# B&R Automation Studio project RobotLineDemo
Automation Studio 6.5.3.11; technology packages: mappMotion 6.9.1, OpcUaCs 6.8.0

## Configuration Config1

CPU 5APC4100.TGL4-000, AutomationRuntime 6.8.1, Build 11.3.0

### Task classes (Cpu.sw)
```
Cyclic#1 (cycle 4000 us, tolerance 0 us):
  MovePrg <- Tasks.MovePrg.prg
Cyclic#2:
  Override <- Tasks.Override.prg
DataObjects: McAcpSys
NcDataObjects: McDriveLog
Binaries: McAcpSim, udbdef, McMechSys, FWRules, McAcpDrv, TCData, Config_19, Config_18, Config_17, Config_16, Config_15, Config_14, arconfig, Config_12, Config_11, Config_10, Config_13, Config_1, ConvAxes, User, Config_4, asfw, iomap, Config_24, Config_23, Config_22, Config_21, UaCsConfig, Config_2, ashwd, Hierarchy, Config_7, ToolGeo, ToolDyn, Config_5, Common, Config, ashwac, sysconf, Config_20, Config_8, ProdLoad1, TrkPaths, Config_9, Config_3, Config_6, BRRole, Config_25
Libraries: MpBase, McBase, MpAxis, McAcpAx, McPathGen, McAxGroup, McAxis, McProgInt, McTrkPath, MpRobotics, ArSvcReg, UaCore, AsIecCon, UaCoal, powerlnk, astime, runtime, fileio, AsIOAcc, SYS_LIB, AsArProf, DataObj, UaCoalPrv, AsIO, brsystem, AsMem, AsIoTrc, AsEPL
```

### Hardware
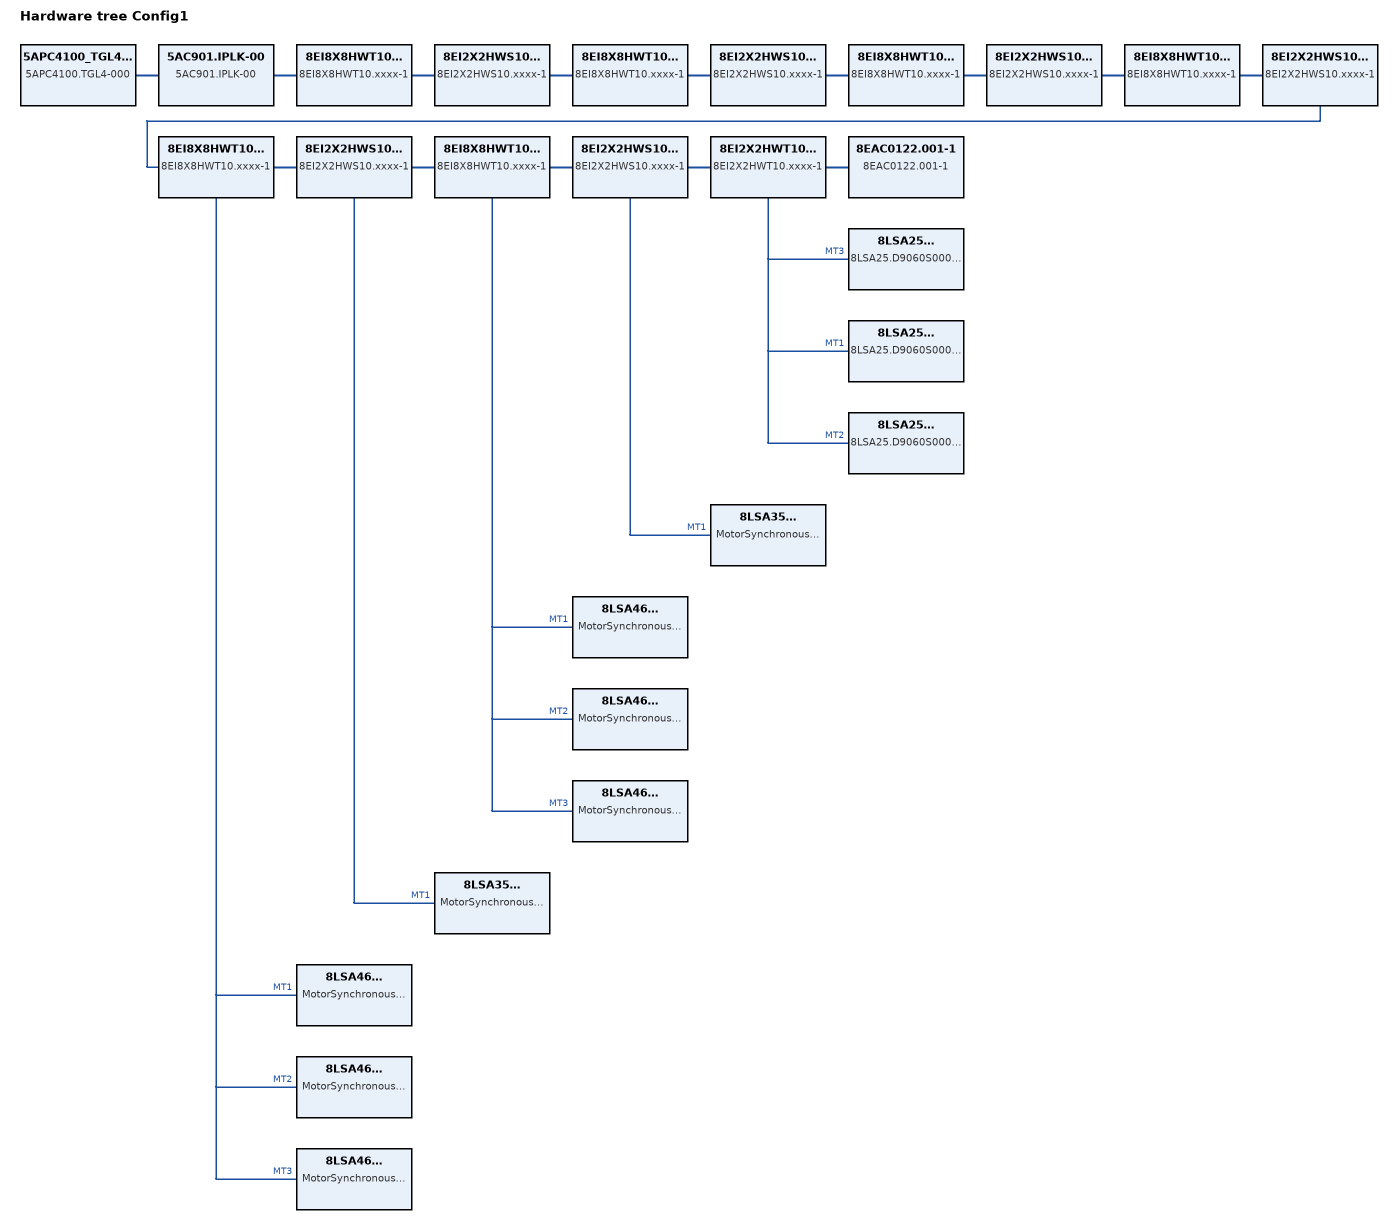
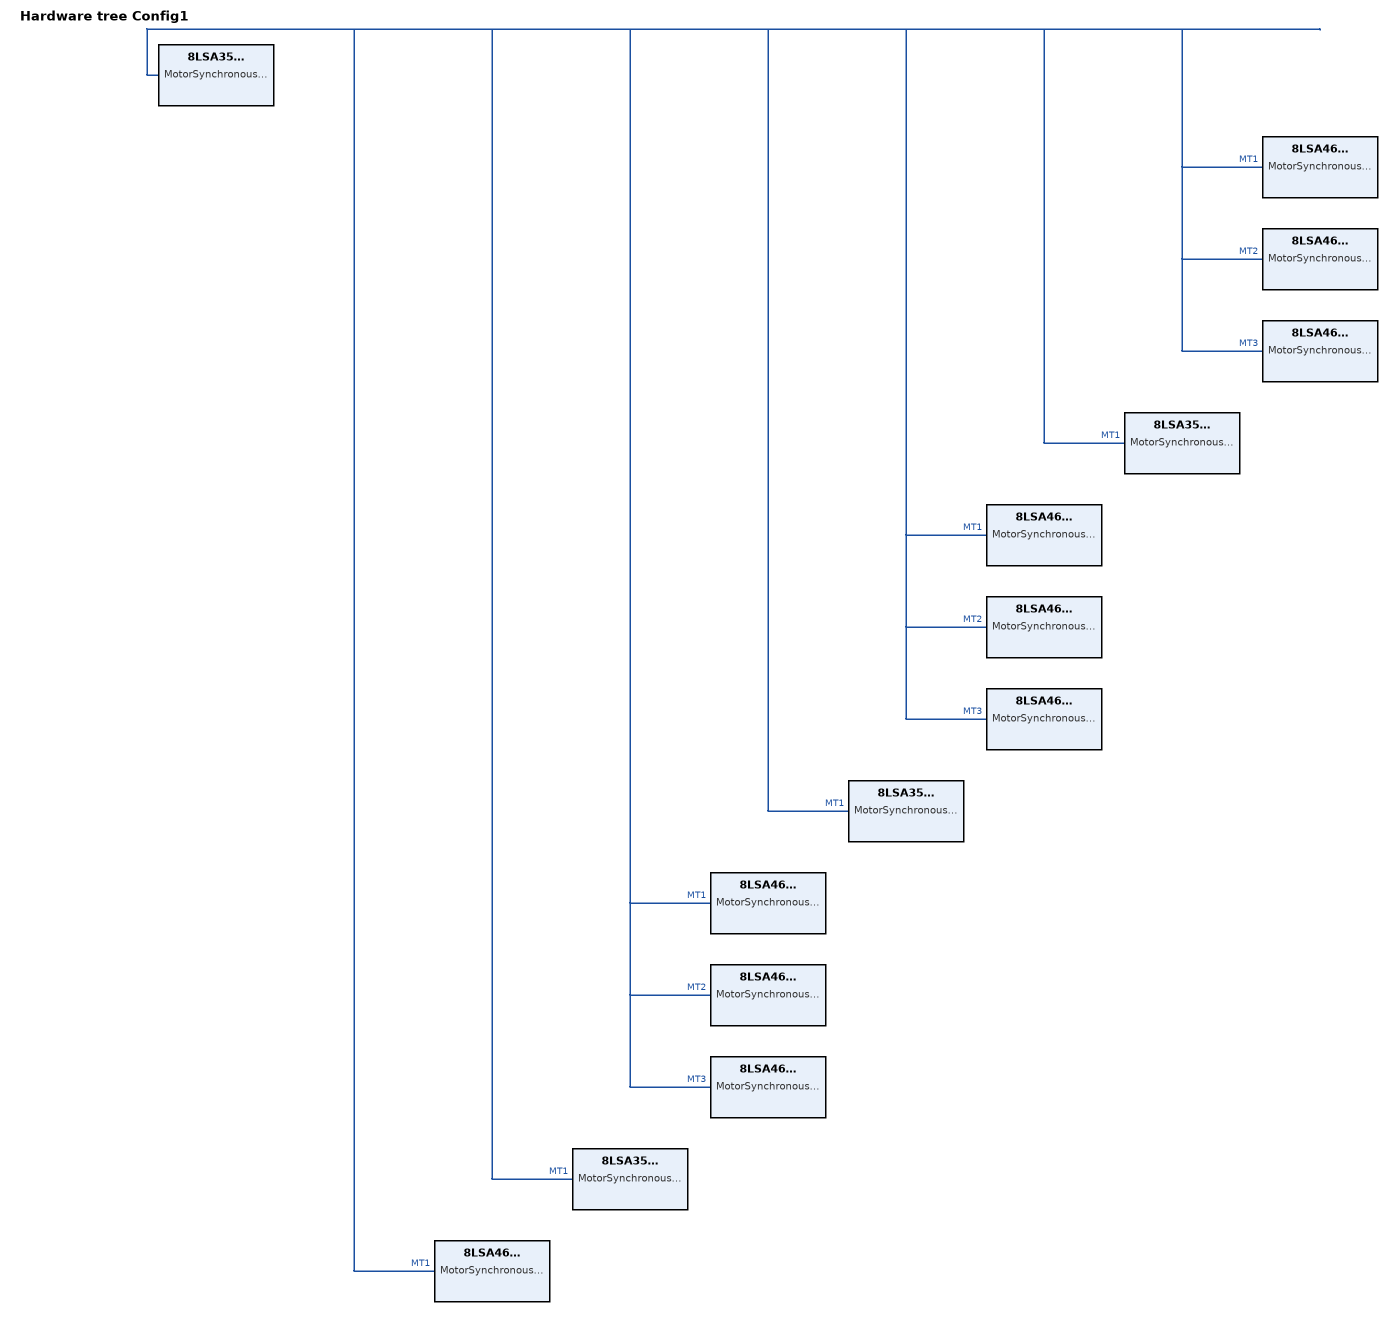
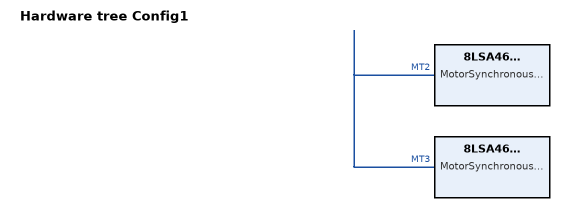
```
5AC901.IPLK-00 : 5AC901.IPLK-00 v2.1.0.0  [SS -> 5APC4100_TGL4_000.SS2]
  Connector IF1:
    EplNatSubnet = 192.168.102.0
5APC4100_TGL4_000 : 5APC4100.TGL4-000 v1.3.1.0
  Connector IF3:
    AssignedOperatingSystem = ARemb
    ActivateDevice = 1
    HostName = laimighoferp-apc4100
    Mode = Manual
    InternetAddress = 172.30.13.10
  Connector IF4:
    AssignedOperatingSystem = ARemb
    ActivateDevice = 1
    HostName = laimighoferp-apc4100
  Connector IF5:
    AssignedOperatingSystem = ARemb
    ActivateDevice = 1
    HostName = laimighoferp-apc4100
  Connector IF6:
    AssignedOperatingSystem = ARemb
    ActivateDevice = 1
    HostName = laimighoferp-apc4100
  Connector IF7:
    AssignedOperatingSystem = ARemb
  Connector IF8:
    AssignedOperatingSystem = ARemb
  Connector IF9:
    AssignedOperatingSystem = ARemb
  Connector IF10:
    AssignedOperatingSystem = ARemb
  Connector IF11:
    AssignedOperatingSystem = ARemb
  Connector IF12:
    AssignedOperatingSystem = ARemb
  ConfigurationID = RobotLineDemoInterpack_Config1
  Simulation = 1
  SimulationIPAddress = 127.0.0.3
  Cyclic1Duration = 4000
  Cyclic1Tolerance = 0
  FileDevice1
  FileDeviceName1 = USER
  FileDevicePath1 = USER_PATH
  FileDevice2
  FileDeviceName2 = CNC_PrgDir
  FileDevicePath2 = USER_PATH/MotionPrg
  FileDevice3
  FileDeviceName3 = Scene
  FileDevicePath3 = USER_PATH/Scenes  // ../../../../../../Logical/Scene/Scenes
  TimeZone = 140
  EthernetHostName = laimighoferp-apc4100
  EthernetDefaultGateway = 172.30.13.1
  ActivateWebServer = 1
  WebServerProtocol = 1
  ActivateSdm = 1
8EAC0122.001-1 : 8EAC0122.001-1 v3.0.0.0  [SS -> 8EI2X2HWT10.xxxx-1.SS1]
8EI2X2HWS10.xxxx-1-QC_D4r1100R_1 : 8EI2X2HWS10.xxxx-1 v2.4.0.0 (NodeNumber=2)  [PLK1 -> 8EI8X8HWT10.xxxx-1-Q1-Q2-Q3_D4r1100R_1.PLK2 [Cable Type=PowerlinkCable, Length=10, Version=1.0.0.3]; PLK2 -> 8EI8X8HWT10.xxxx-1-Q1-Q2-Q3_D4r1100R_2.PLK1 [Cable Type=PowerlinkCable, Length=10, Version=1.0.0.3]]
  DriveConfiguration/Module:
    ActivateACOPOSSimulationOnPLC = 1
  DriveConfiguration/Encoder/EncoderX41:
    InterfaceType = EnDat
  DriveConfiguration/Channel[1]/RealAxis:
    AxisReference = gAxisQC_D4r1100R_1
  DriveConfiguration/Channel[1]/RealAxis/MechanicalElements/Gearbox:
    InputIsReadOnly = 1
    Input = 10
    OutputIsReadOnly = 1
  DriveConfiguration/Channel[1]/RealAxis/MechanicalElements/RotaryToLinearTransformation:
    ReferenceDistanceIsReadOnly = 1
    ReferenceDistance = 360
  DriveConfiguration/Channel[1]/RealAxis/Controller:
    ModeIsReadOnly = 1
    Mode = PositionControllerWithTorqueFeedForward
  DriveConfiguration/Channel[1]/RealAxis/Controller/Mode/Position:
    ProportionalGainIsReadOnly = 1
    ProportionalGain = 25.0
    IntegrationTimeIsReadOnly = 1
  DriveConfiguration/Channel[1]/RealAxis/Controller/Mode/Speed:
    ProportionalGainIsReadOnly = 1
    ProportionalGain = 1.3
    IntegrationTimeIsReadOnly = 1
    FilterTimeIsReadOnly = 1
  DriveConfiguration/Channel[1]/RealAxis/Controller/Mode:
    FeedForwardIsReadOnly = 1
    FeedForward = CyclicValueFromAxesGroup
  DriveConfiguration/Channel[1]/RealAxis/Controller/Mode/LoopFilters:
    LoopFilterXIsReadOnly = 1
  DriveConfiguration/Channel[1]/RealAxis/Homing:
    Mode = Absolute
    RestorePositionVariable = 
  DriveConfiguration/Channel[1]/RealAxis/StopReaction:
    DriveError = CyclicDecelerationFromAxesGroup
  DriveConfiguration/Channel[1]/RealAxis/MovementErrorLimits:
    PositionError = 1.0
  DriveConfiguration/Channel[1]/RealAxis:
    JerkFilterIsReadOnly = 1
    JerkFilter = Used
  DriveConfiguration/Channel[1]/RealAxis/JerkFilter:
    JerkTimeMin = 0.07
    JerkTime = 0.07
8EI2X2HWS10.xxxx-1-QC_D4r1100R_2 : 8EI2X2HWS10.xxxx-1 v2.4.0.0 (NodeNumber=4)  [PLK1 -> 8EI8X8HWT10.xxxx-1-Q1-Q2-Q3_D4r1100R_2.PLK2 [Cable Type=PowerlinkCable, Length=10, Version=1.0.0.3]; PLK2 -> 8EI8X8HWT10.xxxx-1-Q1-Q2-Q3_D4r1100R_3.PLK1 [Cable Type=PowerlinkCable, Length=10, Version=1.0.0.3]]
  DriveConfiguration/Module:
    ActivateACOPOSSimulationOnPLC = 1
  DriveConfiguration/Encoder/EncoderX41:
    InterfaceType = EnDat
  DriveConfiguration/Channel[1]/RealAxis:
    AxisReference = gAxisQC_D4r1100R_2
  DriveConfiguration/Channel[1]/RealAxis/MechanicalElements/Gearbox:
    InputIsReadOnly = 1
    Input = 10
    OutputIsReadOnly = 1
  DriveConfiguration/Channel[1]/RealAxis/MechanicalElements/RotaryToLinearTransformation:
    ReferenceDistanceIsReadOnly = 1
    ReferenceDistance = 360
  DriveConfiguration/Channel[1]/RealAxis/Controller:
    ModeIsReadOnly = 1
    Mode = PositionControllerWithTorqueFeedForward
  DriveConfiguration/Channel[1]/RealAxis/Controller/Mode/Position:
    ProportionalGainIsReadOnly = 1
    ProportionalGain = 25.0
    IntegrationTimeIsReadOnly = 1
  DriveConfiguration/Channel[1]/RealAxis/Controller/Mode/Speed:
    ProportionalGainIsReadOnly = 1
    ProportionalGain = 1.3
    IntegrationTimeIsReadOnly = 1
    FilterTimeIsReadOnly = 1
  DriveConfiguration/Channel[1]/RealAxis/Controller/Mode:
    FeedForwardIsReadOnly = 1
    FeedForward = CyclicValueFromAxesGroup
  DriveConfiguration/Channel[1]/RealAxis/Controller/Mode/LoopFilters:
    LoopFilterXIsReadOnly = 1
  DriveConfiguration/Channel[1]/RealAxis/Homing:
    Mode = Absolute
    RestorePositionVariable = 
  DriveConfiguration/Channel[1]/RealAxis/StopReaction:
    DriveError = CyclicDecelerationFromAxesGroup
  DriveConfiguration/Channel[1]/RealAxis/MovementErrorLimits:
    PositionError = 1.0
  DriveConfiguration/Channel[1]/RealAxis:
    JerkFilterIsReadOnly = 1
    JerkFilter = Used
  DriveConfiguration/Channel[1]/RealAxis/JerkFilter:
    JerkTimeMin = 0.07
    JerkTime = 0.07
8EI2X2HWS10.xxxx-1-QC_D4r1100R_3 : 8EI2X2HWS10.xxxx-1 v2.4.0.0 (NodeNumber=6)  [PLK1 -> 8EI8X8HWT10.xxxx-1-Q1-Q2-Q3_D4r1100R_3.PLK2 [Cable Type=PowerlinkCable, Length=10, Version=1.0.0.3]; PLK2 -> 8EI8X8HWT10.xxxx-1-Q1-Q2-Q3_D4r1100R_4.PLK1 [Cable Type=PowerlinkCable, Length=10, Version=1.0.0.3]]
  DriveConfiguration/Module:
    ActivateACOPOSSimulationOnPLC = 1
  DriveConfiguration/Encoder/EncoderX41:
    InterfaceType = EnDat
  DriveConfiguration/Channel[1]/RealAxis:
    AxisReference = gAxisQC_D4r1100R_3
  DriveConfiguration/Channel[1]/RealAxis/MechanicalElements/Gearbox:
    InputIsReadOnly = 1
    Input = 10
    OutputIsReadOnly = 1
  DriveConfiguration/Channel[1]/RealAxis/MechanicalElements/RotaryToLinearTransformation:
    ReferenceDistanceIsReadOnly = 1
    ReferenceDistance = 360
  DriveConfiguration/Channel[1]/RealAxis/Controller:
    ModeIsReadOnly = 1
    Mode = PositionControllerWithTorqueFeedForward
  DriveConfiguration/Channel[1]/RealAxis/Controller/Mode/Position:
    ProportionalGainIsReadOnly = 1
    ProportionalGain = 25.0
    IntegrationTimeIsReadOnly = 1
  DriveConfiguration/Channel[1]/RealAxis/Controller/Mode/Speed:
    ProportionalGainIsReadOnly = 1
    ProportionalGain = 1.3
    IntegrationTimeIsReadOnly = 1
    FilterTimeIsReadOnly = 1
  DriveConfiguration/Channel[1]/RealAxis/Controller/Mode:
    FeedForwardIsReadOnly = 1
    FeedForward = CyclicValueFromAxesGroup
  DriveConfiguration/Channel[1]/RealAxis/Controller/Mode/LoopFilters:
    LoopFilterXIsReadOnly = 1
  DriveConfiguration/Channel[1]/RealAxis/Homing:
    Mode = Absolute
    RestorePositionVariable = 
  DriveConfiguration/Channel[1]/RealAxis/StopReaction:
    DriveError = CyclicDecelerationFromAxesGroup
  DriveConfiguration/Channel[1]/RealAxis/MovementErrorLimits:
    PositionError = 1.0
  DriveConfiguration/Channel[1]/RealAxis:
    JerkFilterIsReadOnly = 1
    JerkFilter = Used
  DriveConfiguration/Channel[1]/RealAxis/JerkFilter:
    JerkTimeMin = 0.07
    JerkTime = 0.07
8EI2X2HWS10.xxxx-1-QC_D4r1100R_4 : 8EI2X2HWS10.xxxx-1 v2.4.0.0 (NodeNumber=8)  [PLK1 -> 8EI8X8HWT10.xxxx-1-Q1-Q2-Q3_D4r1100R_4.PLK2 [Cable Type=PowerlinkCable, Length=10, Version=1.0.0.3]; PLK2 -> 8EI8X8HWT10.xxxx-1-Q1-Q2-Q3_D4r1100R_5.PLK1 [Cable Type=PowerlinkCable, Length=10, Version=1.0.0.3]]
  DriveConfiguration/Module:
    ActivateACOPOSSimulationOnPLC = 1
  DriveConfiguration/Encoder/EncoderX41:
    InterfaceType = EnDat
  DriveConfiguration/Channel[1]/RealAxis:
    AxisReference = gAxisQC_D4r1100R_4
  DriveConfiguration/Channel[1]/RealAxis/MechanicalElements/Gearbox:
    InputIsReadOnly = 1
    Input = 10
    OutputIsReadOnly = 1
  DriveConfiguration/Channel[1]/RealAxis/MechanicalElements/RotaryToLinearTransformation:
    ReferenceDistanceIsReadOnly = 1
    ReferenceDistance = 360
  DriveConfiguration/Channel[1]/RealAxis/Controller:
    ModeIsReadOnly = 1
    Mode = PositionControllerWithTorqueFeedForward
  DriveConfiguration/Channel[1]/RealAxis/Controller/Mode/Position:
    ProportionalGainIsReadOnly = 1
    ProportionalGain = 25.0
    IntegrationTimeIsReadOnly = 1
  DriveConfiguration/Channel[1]/RealAxis/Controller/Mode/Speed:
    ProportionalGainIsReadOnly = 1
    ProportionalGain = 1.3
    IntegrationTimeIsReadOnly = 1
    FilterTimeIsReadOnly = 1
  DriveConfiguration/Channel[1]/RealAxis/Controller/Mode:
    FeedForwardIsReadOnly = 1
    FeedForward = CyclicValueFromAxesGroup
  DriveConfiguration/Channel[1]/RealAxis/Controller/Mode/LoopFilters:
    LoopFilterXIsReadOnly = 1
  DriveConfiguration/Channel[1]/RealAxis/Homing:
    Mode = Absolute
    RestorePositionVariable = 
  DriveConfiguration/Channel[1]/RealAxis/StopReaction:
    DriveError = CyclicDecelerationFromAxesGroup
  DriveConfiguration/Channel[1]/RealAxis/MovementErrorLimits:
    PositionError = 1.0
  DriveConfiguration/Channel[1]/RealAxis:
    JerkFilterIsReadOnly = 1
    JerkFilter = Used
  DriveConfiguration/Channel[1]/RealAxis/JerkFilter:
    JerkTimeMin = 0.07
    JerkTime = 0.07
8EI2X2HWS10.xxxx-1-QC_D4r1100R_5 : 8EI2X2HWS10.xxxx-1 v2.4.0.0 (NodeNumber=10)  [PLK1 -> 8EI8X8HWT10.xxxx-1-Q1-Q2-Q3_D4r1100R_5.PLK2 [Cable Type=PowerlinkCable, Length=10, Version=1.0.0.3]; PLK2 -> 8EI8X8HWT10.xxxx-1-Q1-Q2-Q3_D4r1100R_6.PLK1 [Cable Type=PowerlinkCable, Length=10, Version=1.0.0.3]]
  DriveConfiguration/Module:
    ActivateACOPOSSimulationOnPLC = 1
  DriveConfiguration/Encoder/EncoderX41:
    InterfaceType = EnDat
  DriveConfiguration/Channel[1]/RealAxis:
    AxisReference = gAxisQC_D4r1100R_5
  DriveConfiguration/Channel[1]/RealAxis/MechanicalElements/Gearbox:
    InputIsReadOnly = 1
    Input = 10
    OutputIsReadOnly = 1
  DriveConfiguration/Channel[1]/RealAxis/MechanicalElements/RotaryToLinearTransformation:
    ReferenceDistanceIsReadOnly = 1
    ReferenceDistance = 360
  DriveConfiguration/Channel[1]/RealAxis/Controller:
    ModeIsReadOnly = 1
    Mode = PositionControllerWithTorqueFeedForward
  DriveConfiguration/Channel[1]/RealAxis/Controller/Mode/Position:
    ProportionalGainIsReadOnly = 1
    ProportionalGain = 25.0
    IntegrationTimeIsReadOnly = 1
  DriveConfiguration/Channel[1]/RealAxis/Controller/Mode/Speed:
    ProportionalGainIsReadOnly = 1
    ProportionalGain = 1.3
    IntegrationTimeIsReadOnly = 1
    FilterTimeIsReadOnly = 1
  DriveConfiguration/Channel[1]/RealAxis/Controller/Mode:
    FeedForwardIsReadOnly = 1
    FeedForward = CyclicValueFromAxesGroup
  DriveConfiguration/Channel[1]/RealAxis/Controller/Mode/LoopFilters:
    LoopFilterXIsReadOnly = 1
  DriveConfiguration/Channel[1]/RealAxis/Homing:
    Mode = Absolute
    RestorePositionVariable = 
  DriveConfiguration/Channel[1]/RealAxis/StopReaction:
    DriveError = CyclicDecelerationFromAxesGroup
  DriveConfiguration/Channel[1]/RealAxis/MovementErrorLimits:
    PositionError = 1.0
  DriveConfiguration/Channel[1]/RealAxis:
    JerkFilterIsReadOnly = 1
    JerkFilter = Used
  DriveConfiguration/Channel[1]/RealAxis/JerkFilter:
    JerkTimeMin = 0.07
    JerkTime = 0.07
8EI2X2HWS10.xxxx-1-QC_D4r1100R_6 : 8EI2X2HWS10.xxxx-1 v2.4.0.0 (NodeNumber=12)  [PLK1 -> 8EI8X8HWT10.xxxx-1-Q1-Q2-Q3_D4r1100R_6.PLK2 [Cable Type=PowerlinkCable, Length=10, Version=1.0.0.3]; PLK2 -> 8EI2X2HWT10.xxxx-1.PLK1 [Cable Type=PowerlinkCable, Length=10, Version=1.0.0.3]]
  DriveConfiguration/Module:
    ActivateACOPOSSimulationOnPLC = 1
  DriveConfiguration/Encoder/EncoderX41:
    InterfaceType = EnDat
  DriveConfiguration/Channel[1]/RealAxis:
    AxisReference = gAxisQC_D4r1100R_6
  DriveConfiguration/Channel[1]/RealAxis/MechanicalElements/Gearbox:
    InputIsReadOnly = 1
    Input = 10
    OutputIsReadOnly = 1
  DriveConfiguration/Channel[1]/RealAxis/MechanicalElements/RotaryToLinearTransformation:
    ReferenceDistanceIsReadOnly = 1
    ReferenceDistance = 360
  DriveConfiguration/Channel[1]/RealAxis/Controller:
    ModeIsReadOnly = 1
    Mode = PositionControllerWithTorqueFeedForward
  DriveConfiguration/Channel[1]/RealAxis/Controller/Mode/Position:
    ProportionalGainIsReadOnly = 1
    ProportionalGain = 25.0
    IntegrationTimeIsReadOnly = 1
  DriveConfiguration/Channel[1]/RealAxis/Controller/Mode/Speed:
    ProportionalGainIsReadOnly = 1
    ProportionalGain = 1.3
    IntegrationTimeIsReadOnly = 1
    FilterTimeIsReadOnly = 1
  DriveConfiguration/Channel[1]/RealAxis/Controller/Mode:
    FeedForwardIsReadOnly = 1
    FeedForward = CyclicValueFromAxesGroup
  DriveConfiguration/Channel[1]/RealAxis/Controller/Mode/LoopFilters:
    LoopFilterXIsReadOnly = 1
  DriveConfiguration/Channel[1]/RealAxis/Homing:
    Mode = Absolute
    RestorePositionVariable = 
  DriveConfiguration/Channel[1]/RealAxis/StopReaction:
    DriveError = CyclicDecelerationFromAxesGroup
  DriveConfiguration/Channel[1]/RealAxis/MovementErrorLimits:
    PositionError = 1.0
  DriveConfiguration/Channel[1]/RealAxis:
    JerkFilterIsReadOnly = 1
    JerkFilter = Used
  DriveConfiguration/Channel[1]/RealAxis/JerkFilter:
    JerkTimeMin = 0.07
    JerkTime = 0.07
8EI2X2HWT10.xxxx-1 : 8EI2X2HWT10.xxxx-1 v2.4.0.0 (NodeNumber=13)  [PLK1 -> 8EI2X2HWS10.xxxx-1-QC_D4r1100R_6.PLK2 [Cable Type=PowerlinkCable, Length=10, Version=1.0.0.3]; MT2 -> 8LSA25.D9060S000-3_b.MT; MT3 -> 8LSA25.D9060S000-3.MT]
  DriveConfiguration/Module:
    ActivateACOPOSSimulationOnPLC = 1
  DriveConfiguration/Channel[1]/RealAxis:
    AxisReference = gAxis_Conveyor_1
  DriveConfiguration/Channel[2]/RealAxis:
    AxisReference = gAxis_Conveyor_2
8EI8X8HWT10.xxxx-1-Q1-Q2-Q3_D4r1100R_1 : 8EI8X8HWT10.xxxx-1 v2.4.0.0 (NodeNumber=1)  [PLK1 -> 5AC901.IPLK-00.IF1 [Cable Type=PowerlinkCable, Length=10, Version=1.0.0.3]; PLK2 -> 8EI2X2HWS10.xxxx-1-QC_D4r1100R_1.PLK1 [Cable Type=PowerlinkCable, Length=10, Version=1.0.0.3]; MT2 -> 8LSA46.DB060S200-3-Q2_D4r1100R_1.MT; MT3 -> 8LSA46.DB060S200-3-Q3_D4r1100R_1.MT]
  DriveConfiguration/Module:
    ActivateACOPOSSimulationOnPLC = 1
  DriveConfiguration/Encoder/EncoderX41:
    InterfaceType = EnDat
  DriveConfiguration/Encoder/EncoderX42:
    InterfaceType = EnDat
  DriveConfiguration/Encoder/EncoderX43:
    InterfaceType = EnDat
  DriveConfiguration/Channel[1]/RealAxis:
    AxisReference = gAxisQ1_D4r1100R_1
  DriveConfiguration/Channel[1]/RealAxis/MechanicalElements/Gearbox:
    InputIsReadOnly = 1
    Input = 77
    OutputIsReadOnly = 1
    Output = 2
  DriveConfiguration/Channel[1]/RealAxis/MechanicalElements/RotaryToLinearTransformation:
    ReferenceDistanceIsReadOnly = 1
    ReferenceDistance = 360
  DriveConfiguration/Channel[1]/RealAxis/Controller:
    ModeIsReadOnly = 1
    Mode = PositionControllerWithTorqueFeedForward
  DriveConfiguration/Channel[1]/RealAxis/Controller/Mode/Position:
    ProportionalGainIsReadOnly = 1
    ProportionalGain = 15.0
    IntegrationTimeIsReadOnly = 1
  DriveConfiguration/Channel[1]/RealAxis/Controller/Mode/Speed:
    ProportionalGainIsReadOnly = 1
    ProportionalGain = 8.0
    IntegrationTimeIsReadOnly = 1
    FilterTimeIsReadOnly = 1
  DriveConfiguration/Channel[1]/RealAxis/Controller/Mode:
    FeedForwardIsReadOnly = 1
    FeedForward = CyclicValueFromAxesGroup
  DriveConfiguration/Channel[1]/RealAxis/Controller/Mode/LoopFilters:
    LoopFilterXIsReadOnly = 1
  DriveConfiguration/Channel[1]/RealAxis/Homing:
    Mode = AbsoluteCorrection
    RestorePositionVariable = 
  DriveConfiguration/Channel[1]/RealAxis/StopReaction:
    DriveError = CyclicDecelerationFromAxesGroup
  DriveConfiguration/Channel[1]/RealAxis/MovementErrorLimits:
    PositionError = 0.5
  DriveConfiguration/Channel[1]/RealAxis:
    JerkFilterIsReadOnly = 1
    JerkFilter = Used
  DriveConfiguration/Channel[1]/RealAxis/JerkFilter:
    JerkTimeMin = 0.07
    JerkTime = 0.07
  DriveConfiguration/Channel[2]/RealAxis:
    AxisReference = gAxisQ2_D4r1100R_1
  DriveConfiguration/Channel[2]/RealAxis/MechanicalElements/Gearbox:
    InputIsReadOnly = 1
    Input = 77
    OutputIsReadOnly = 1
    Output = 2
  DriveConfiguration/Channel[2]/RealAxis/MechanicalElements/RotaryToLinearTransformation:
    ReferenceDistanceIsReadOnly = 1
    ReferenceDistance = 360
  DriveConfiguration/Channel[2]/RealAxis/Controller:
    ModeIsReadOnly = 1
    Mode = PositionControllerWithTorqueFeedForward
  DriveConfiguration/Channel[2]/RealAxis/Controller/Mode/Position:
    ProportionalGainIsReadOnly = 1
    ProportionalGain = 15.0
    IntegrationTimeIsReadOnly = 1
  DriveConfiguration/Channel[2]/RealAxis/Controller/Mode/Speed:
    ProportionalGainIsReadOnly = 1
    ProportionalGain = 8.0
    IntegrationTimeIsReadOnly = 1
    FilterTimeIsReadOnly = 1
  DriveConfiguration/Channel[2]/RealAxis/Controller/Mode:
    FeedForwardIsReadOnly = 1
    FeedForward = CyclicValueFromAxesGroup
  DriveConfiguration/Channel[2]/RealAxis/Controller/Mode/LoopFilters:
    LoopFilterXIsReadOnly = 1
  DriveConfiguration/Channel[2]/RealAxis/Homing:
    Mode = AbsoluteCorrection
    RestorePositionVariable = 
  DriveConfiguration/Channel[2]/RealAxis/StopReaction:
    DriveError = CyclicDecelerationFromAxesGroup
  DriveConfiguration/Channel[2]/RealAxis/MovementErrorLimits:
    PositionError = 0.5
  DriveConfiguration/Channel[2]/RealAxis:
    JerkFilterIsReadOnly = 1
    JerkFilter = Used
  DriveConfiguration/Channel[2]/RealAxis/JerkFilter:
    JerkTimeMin = 0.07
    JerkTime = 0.07
  DriveConfiguration/Channel[3]/RealAxis:
    AxisReference = gAxisQ3_D4r1100R_1
  DriveConfiguration/Channel[3]/RealAxis/MechanicalElements/Gearbox:
    InputIsReadOnly = 1
    Input = 77
    OutputIsReadOnly = 1
    Output = 2
  DriveConfiguration/Channel[3]/RealAxis/MechanicalElements/RotaryToLinearTransformation:
    ReferenceDistanceIsReadOnly = 1
    ReferenceDistance = 360
  DriveConfiguration/Channel[3]/RealAxis/Controller:
    ModeIsReadOnly = 1
    Mode = PositionControllerWithTorqueFeedForward
  DriveConfiguration/Channel[3]/RealAxis/Controller/Mode/Position:
    ProportionalGainIsReadOnly = 1
    ProportionalGain = 15.0
    IntegrationTimeIsReadOnly = 1
  DriveConfiguration/Channel[3]/RealAxis/Controller/Mode/Speed:
    ProportionalGainIsReadOnly = 1
    ProportionalGain = 8.0
    IntegrationTimeIsReadOnly = 1
    FilterTimeIsReadOnly = 1
  DriveConfiguration/Channel[3]/RealAxis/Controller/Mode:
    FeedForwardIsReadOnly = 1
    FeedForward = CyclicValueFromAxesGroup
  DriveConfiguration/Channel[3]/RealAxis/Controller/Mode/LoopFilters:
    LoopFilterXIsReadOnly = 1
  DriveConfiguration/Channel[3]/RealAxis/Homing:
    Mode = AbsoluteCorrection
    RestorePositionVariable = 
  DriveConfiguration/Channel[3]/RealAxis/StopReaction:
    DriveError = CyclicDecelerationFromAxesGroup
  DriveConfiguration/Channel[3]/RealAxis/MovementErrorLimits:
    PositionError = 0.5
  DriveConfiguration/Channel[3]/RealAxis:
    JerkFilterIsReadOnly = 1
    JerkFilter = Used
  DriveConfiguration/Channel[3]/RealAxis/JerkFilter:
    JerkTimeMin = 0.07
    JerkTime = 0.07
8EI8X8HWT10.xxxx-1-Q1-Q2-Q3_D4r1100R_2 : 8EI8X8HWT10.xxxx-1 v2.4.0.0 (NodeNumber=3)  [PLK1 -> 8EI2X2HWS10.xxxx-1-QC_D4r1100R_1.PLK2 [Cable Type=PowerlinkCable, Length=10, Version=1.0.0.3]; PLK2 -> 8EI2X2HWS10.xxxx-1-QC_D4r1100R_2.PLK1 [Cable Type=PowerlinkCable, Length=10, Version=1.0.0.3]; MT2 -> 8LSA46.DB060S200-3-Q2_D4r1100R_2.MT; MT3 -> 8LSA46.DB060S200-3-Q3_D4r1100R_2.MT]
  DriveConfiguration/Module:
    ActivateACOPOSSimulationOnPLC = 1
  DriveConfiguration/Encoder/EncoderX41:
    InterfaceType = EnDat
  DriveConfiguration/Encoder/EncoderX42:
    InterfaceType = EnDat
  DriveConfiguration/Encoder/EncoderX43:
    InterfaceType = EnDat
  DriveConfiguration/Channel[1]/RealAxis:
    AxisReference = gAxisQ1_D4r1100R_2
  DriveConfiguration/Channel[1]/RealAxis/MechanicalElements/Gearbox:
    InputIsReadOnly = 1
    Input = 77
    OutputIsReadOnly = 1
    Output = 2
  DriveConfiguration/Channel[1]/RealAxis/MechanicalElements/RotaryToLinearTransformation:
    ReferenceDistanceIsReadOnly = 1
    ReferenceDistance = 360
  DriveConfiguration/Channel[1]/RealAxis/Controller:
    ModeIsReadOnly = 1
    Mode = PositionControllerWithTorqueFeedForward
  DriveConfiguration/Channel[1]/RealAxis/Controller/Mode/Position:
    ProportionalGainIsReadOnly = 1
    ProportionalGain = 15.0
    IntegrationTimeIsReadOnly = 1
  DriveConfiguration/Channel[1]/RealAxis/Controller/Mode/Speed:
    ProportionalGainIsReadOnly = 1
    ProportionalGain = 8.0
    IntegrationTimeIsReadOnly = 1
    FilterTimeIsReadOnly = 1
  DriveConfiguration/Channel[1]/RealAxis/Controller/Mode:
    FeedForwardIsReadOnly = 1
    FeedForward = CyclicValueFromAxesGroup
  DriveConfiguration/Channel[1]/RealAxis/Controller/Mode/LoopFilters:
    LoopFilterXIsReadOnly = 1
  DriveConfiguration/Channel[1]/RealAxis/Homing:
    Mode = AbsoluteCorrection
    RestorePositionVariable = 
  DriveConfiguration/Channel[1]/RealAxis/StopReaction:
    DriveError = CyclicDecelerationFromAxesGroup
  DriveConfiguration/Channel[1]/RealAxis/MovementErrorLimits:
    PositionError = 0.5
  DriveConfiguration/Channel[1]/RealAxis:
    JerkFilterIsReadOnly = 1
    JerkFilter = Used
  DriveConfiguration/Channel[1]/RealAxis/JerkFilter:
    JerkTimeMin = 0.07
    JerkTime = 0.07
  DriveConfiguration/Channel[2]/RealAxis:
    AxisReference = gAxisQ2_D4r1100R_2
  DriveConfiguration/Channel[2]/RealAxis/MechanicalElements/Gearbox:
    InputIsReadOnly = 1
    Input = 77
    OutputIsReadOnly = 1
    Output = 2
  DriveConfiguration/Channel[2]/RealAxis/MechanicalElements/RotaryToLinearTransformation:
    ReferenceDistanceIsReadOnly = 1
    ReferenceDistance = 360
  DriveConfiguration/Channel[2]/RealAxis/Controller:
    ModeIsReadOnly = 1
    Mode = PositionControllerWithTorqueFeedForward
  DriveConfiguration/Channel[2]/RealAxis/Controller/Mode/Position:
    ProportionalGainIsReadOnly = 1
    ProportionalGain = 15.0
    IntegrationTimeIsReadOnly = 1
  DriveConfiguration/Channel[2]/RealAxis/Controller/Mode/Speed:
    ProportionalGainIsReadOnly = 1
    ProportionalGain = 8.0
    IntegrationTimeIsReadOnly = 1
    FilterTimeIsReadOnly = 1
  DriveConfiguration/Channel[2]/RealAxis/Controller/Mode:
    FeedForwardIsReadOnly = 1
    FeedForward = CyclicValueFromAxesGroup
  DriveConfiguration/Channel[2]/RealAxis/Controller/Mode/LoopFilters:
    LoopFilterXIsReadOnly = 1
  DriveConfiguration/Channel[2]/RealAxis/Homing:
    Mode = AbsoluteCorrection
    RestorePositionVariable = 
  DriveConfiguration/Channel[2]/RealAxis/StopReaction:
    DriveError = CyclicDecelerationFromAxesGroup
  DriveConfiguration/Channel[2]/RealAxis/MovementErrorLimits:
    PositionError = 0.5
  DriveConfiguration/Channel[2]/RealAxis:
    JerkFilterIsReadOnly = 1
    JerkFilter = Used
  DriveConfiguration/Channel[2]/RealAxis/JerkFilter:
    JerkTimeMin = 0.07
    JerkTime = 0.07
  DriveConfiguration/Channel[3]/RealAxis:
    AxisReference = gAxisQ3_D4r1100R_2
  DriveConfiguration/Channel[3]/RealAxis/MechanicalElements/Gearbox:
    InputIsReadOnly = 1
    Input = 77
    OutputIsReadOnly = 1
    Output = 2
  DriveConfiguration/Channel[3]/RealAxis/MechanicalElements/RotaryToLinearTransformation:
    ReferenceDistanceIsReadOnly = 1
    ReferenceDistance = 360
  DriveConfiguration/Channel[3]/RealAxis/Controller:
    ModeIsReadOnly = 1
    Mode = PositionControllerWithTorqueFeedForward
  DriveConfiguration/Channel[3]/RealAxis/Controller/Mode/Position:
    ProportionalGainIsReadOnly = 1
    ProportionalGain = 15.0
    IntegrationTimeIsReadOnly = 1
  DriveConfiguration/Channel[3]/RealAxis/Controller/Mode/Speed:
    ProportionalGainIsReadOnly = 1
    ProportionalGain = 8.0
    IntegrationTimeIsReadOnly = 1
    FilterTimeIsReadOnly = 1
  DriveConfiguration/Channel[3]/RealAxis/Controller/Mode:
    FeedForwardIsReadOnly = 1
    FeedForward = CyclicValueFromAxesGroup
  DriveConfiguration/Channel[3]/RealAxis/Controller/Mode/LoopFilters:
    LoopFilterXIsReadOnly = 1
  DriveConfiguration/Channel[3]/RealAxis/Homing:
    Mode = AbsoluteCorrection
    RestorePositionVariable = 
  DriveConfiguration/Channel[3]/RealAxis/StopReaction:
    DriveError = CyclicDecelerationFromAxesGroup
  DriveConfiguration/Channel[3]/RealAxis/MovementErrorLimits:
    PositionError = 0.5
  DriveConfiguration/Channel[3]/RealAxis:
    JerkFilterIsReadOnly = 1
    JerkFilter = Used
  DriveConfiguration/Channel[3]/RealAxis/JerkFilter:
    JerkTimeMin = 0.07
    JerkTime = 0.07
8EI8X8HWT10.xxxx-1-Q1-Q2-Q3_D4r1100R_3 : 8EI8X8HWT10.xxxx-1 v2.4.0.0 (NodeNumber=5)  [PLK1 -> 8EI2X2HWS10.xxxx-1-QC_D4r1100R_2.PLK2 [Cable Type=PowerlinkCable, Length=10, Version=1.0.0.3]; PLK2 -> 8EI2X2HWS10.xxxx-1-QC_D4r1100R_3.PLK1 [Cable Type=PowerlinkCable, Length=10, Version=1.0.0.3]; MT2 -> 8LSA46.DB060S200-3-Q2_D4r1100R_3.MT; MT3 -> 8LSA46.DB060S200-3-Q3_D4r1100R_3.MT]
  DriveConfiguration/Module:
    ActivateACOPOSSimulationOnPLC = 1
  DriveConfiguration/Encoder/EncoderX41:
    InterfaceType = EnDat
  DriveConfiguration/Encoder/EncoderX42:
    InterfaceType = EnDat
  DriveConfiguration/Encoder/EncoderX43:
    InterfaceType = EnDat
  DriveConfiguration/Channel[1]/RealAxis:
    AxisReference = gAxisQ1_D4r1100R_3
  DriveConfiguration/Channel[1]/RealAxis/MechanicalElements/Gearbox:
    InputIsReadOnly = 1
    Input = 77
    OutputIsReadOnly = 1
    Output = 2
  DriveConfiguration/Channel[1]/RealAxis/MechanicalElements/RotaryToLinearTransformation:
    ReferenceDistanceIsReadOnly = 1
    ReferenceDistance = 360
  DriveConfiguration/Channel[1]/RealAxis/Controller:
    ModeIsReadOnly = 1
    Mode = PositionControllerWithTorqueFeedForward
  DriveConfiguration/Channel[1]/RealAxis/Controller/Mode/Position:
    ProportionalGainIsReadOnly = 1
    ProportionalGain = 15.0
    IntegrationTimeIsReadOnly = 1
  DriveConfiguration/Channel[1]/RealAxis/Controller/Mode/Speed:
    ProportionalGainIsReadOnly = 1
    ProportionalGain = 8.0
    IntegrationTimeIsReadOnly = 1
    FilterTimeIsReadOnly = 1
  DriveConfiguration/Channel[1]/RealAxis/Controller/Mode:
    FeedForwardIsReadOnly = 1
    FeedForward = CyclicValueFromAxesGroup
  DriveConfiguration/Channel[1]/RealAxis/Controller/Mode/LoopFilters:
    LoopFilterXIsReadOnly = 1
  DriveConfiguration/Channel[1]/RealAxis/Homing:
    Mode = AbsoluteCorrection
    RestorePositionVariable = 
  DriveConfiguration/Channel[1]/RealAxis/StopReaction:
    DriveError = CyclicDecelerationFromAxesGroup
  DriveConfiguration/Channel[1]/RealAxis/MovementErrorLimits:
    PositionError = 0.5
  DriveConfiguration/Channel[1]/RealAxis:
    JerkFilterIsReadOnly = 1
    JerkFilter = Used
  DriveConfiguration/Channel[1]/RealAxis/JerkFilter:
    JerkTimeMin = 0.07
    JerkTime = 0.07
  DriveConfiguration/Channel[2]/RealAxis:
    AxisReference = gAxisQ2_D4r1100R_3
  DriveConfiguration/Channel[2]/RealAxis/MechanicalElements/Gearbox:
    InputIsReadOnly = 1
    Input = 77
    OutputIsReadOnly = 1
    Output = 2
  DriveConfiguration/Channel[2]/RealAxis/MechanicalElements/RotaryToLinearTransformation:
    ReferenceDistanceIsReadOnly = 1
    ReferenceDistance = 360
  DriveConfiguration/Channel[2]/RealAxis/Controller:
    ModeIsReadOnly = 1
    Mode = PositionControllerWithTorqueFeedForward
  DriveConfiguration/Channel[2]/RealAxis/Controller/Mode/Position:
    ProportionalGainIsReadOnly = 1
    ProportionalGain = 15.0
    IntegrationTimeIsReadOnly = 1
  DriveConfiguration/Channel[2]/RealAxis/Controller/Mode/Speed:
    ProportionalGainIsReadOnly = 1
    ProportionalGain = 8.0
    IntegrationTimeIsReadOnly = 1
    FilterTimeIsReadOnly = 1
  DriveConfiguration/Channel[2]/RealAxis/Controller/Mode:
    FeedForwardIsReadOnly = 1
    FeedForward = CyclicValueFromAxesGroup
  DriveConfiguration/Channel[2]/RealAxis/Controller/Mode/LoopFilters:
    LoopFilterXIsReadOnly = 1
  DriveConfiguration/Channel[2]/RealAxis/Homing:
    Mode = AbsoluteCorrection
    RestorePositionVariable = 
  DriveConfiguration/Channel[2]/RealAxis/StopReaction:
    DriveError = CyclicDecelerationFromAxesGroup
  DriveConfiguration/Channel[2]/RealAxis/MovementErrorLimits:
    PositionError = 0.5
  DriveConfiguration/Channel[2]/RealAxis:
    JerkFilterIsReadOnly = 1
    JerkFilter = Used
  DriveConfiguration/Channel[2]/RealAxis/JerkFilter:
    JerkTimeMin = 0.07
    JerkTime = 0.07
  DriveConfiguration/Channel[3]/RealAxis:
    AxisReference = gAxisQ3_D4r1100R_3
  DriveConfiguration/Channel[3]/RealAxis/MechanicalElements/Gearbox:
    InputIsReadOnly = 1
    Input = 77
    OutputIsReadOnly = 1
    Output = 2
  DriveConfiguration/Channel[3]/RealAxis/MechanicalElements/RotaryToLinearTransformation:
    ReferenceDistanceIsReadOnly = 1
    ReferenceDistance = 360
  DriveConfiguration/Channel[3]/RealAxis/Controller:
    ModeIsReadOnly = 1
    Mode = PositionControllerWithTorqueFeedForward
  DriveConfiguration/Channel[3]/RealAxis/Controller/Mode/Position:
    ProportionalGainIsReadOnly = 1
    ProportionalGain = 15.0
    IntegrationTimeIsReadOnly = 1
  DriveConfiguration/Channel[3]/RealAxis/Controller/Mode/Speed:
    ProportionalGainIsReadOnly = 1
    ProportionalGain = 8.0
    IntegrationTimeIsReadOnly = 1
    FilterTimeIsReadOnly = 1
  DriveConfiguration/Channel[3]/RealAxis/Controller/Mode:
    FeedForwardIsReadOnly = 1
    FeedForward = CyclicValueFromAxesGroup
  DriveConfiguration/Channel[3]/RealAxis/Controller/Mode/LoopFilters:
    LoopFilterXIsReadOnly = 1
  DriveConfiguration/Channel[3]/RealAxis/Homing:
    Mode = AbsoluteCorrection
    RestorePositionVariable = 
  DriveConfiguration/Channel[3]/RealAxis/StopReaction:
    DriveError = CyclicDecelerationFromAxesGroup
  DriveConfiguration/Channel[3]/RealAxis/MovementErrorLimits:
    PositionError = 0.5
  DriveConfiguration/Channel[3]/RealAxis:
    JerkFilterIsReadOnly = 1
    JerkFilter = Used
  DriveConfiguration/Channel[3]/RealAxis/JerkFilter:
    JerkTimeMin = 0.07
    JerkTime = 0.07
8EI8X8HWT10.xxxx-1-Q1-Q2-Q3_D4r1100R_4 : 8EI8X8HWT10.xxxx-1 v2.4.0.0 (NodeNumber=7)  [PLK1 -> 8EI2X2HWS10.xxxx-1-QC_D4r1100R_3.PLK2 [Cable Type=PowerlinkCable, Length=10, Version=1.0.0.3]; PLK2 -> 8EI2X2HWS10.xxxx-1-QC_D4r1100R_4.PLK1 [Cable Type=PowerlinkCable, Length=10, Version=1.0.0.3]; MT2 -> 8LSA46.DB060S200-3-Q2_D4r1100R_4.MT; MT3 -> 8LSA46.DB060S200-3-Q3_D4r1100R_4.MT]
  DriveConfiguration/Module:
    ActivateACOPOSSimulationOnPLC = 1
  DriveConfiguration/Encoder/EncoderX41:
    InterfaceType = EnDat
  DriveConfiguration/Encoder/EncoderX42:
    InterfaceType = EnDat
  DriveConfiguration/Encoder/EncoderX43:
    InterfaceType = EnDat
  DriveConfiguration/Channel[1]/RealAxis:
    AxisReference = gAxisQ1_D4r1100R_4
  DriveConfiguration/Channel[1]/RealAxis/MechanicalElements/Gearbox:
    InputIsReadOnly = 1
    Input = 77
    OutputIsReadOnly = 1
    Output = 2
  DriveConfiguration/Channel[1]/RealAxis/MechanicalElements/RotaryToLinearTransformation:
    ReferenceDistanceIsReadOnly = 1
    ReferenceDistance = 360
  DriveConfiguration/Channel[1]/RealAxis/Controller:
    ModeIsReadOnly = 1
    Mode = PositionControllerWithTorqueFeedForward
  DriveConfiguration/Channel[1]/RealAxis/Controller/Mode/Position:
    ProportionalGainIsReadOnly = 1
    ProportionalGain = 15.0
    IntegrationTimeIsReadOnly = 1
  DriveConfiguration/Channel[1]/RealAxis/Controller/Mode/Speed:
    ProportionalGainIsReadOnly = 1
    ProportionalGain = 8.0
    IntegrationTimeIsReadOnly = 1
    FilterTimeIsReadOnly = 1
  DriveConfiguration/Channel[1]/RealAxis/Controller/Mode:
    FeedForwardIsReadOnly = 1
    FeedForward = CyclicValueFromAxesGroup
  DriveConfiguration/Channel[1]/RealAxis/Controller/Mode/LoopFilters:
    LoopFilterXIsReadOnly = 1
  DriveConfiguration/Channel[1]/RealAxis/Homing:
    Mode = AbsoluteCorrection
    RestorePositionVariable = 
  DriveConfiguration/Channel[1]/RealAxis/StopReaction:
    DriveError = CyclicDecelerationFromAxesGroup
  DriveConfiguration/Channel[1]/RealAxis/MovementErrorLimits:
    PositionError = 0.5
  DriveConfiguration/Channel[1]/RealAxis:
    JerkFilterIsReadOnly = 1
    JerkFilter = Used
  DriveConfiguration/Channel[1]/RealAxis/JerkFilter:
    JerkTimeMin = 0.07
    JerkTime = 0.07
  DriveConfiguration/Channel[2]/RealAxis:
    AxisReference = gAxisQ2_D4r1100R_4
  DriveConfiguration/Channel[2]/RealAxis/MechanicalElements/Gearbox:
    InputIsReadOnly = 1
    Input = 77
    OutputIsReadOnly = 1
    Output = 2
  DriveConfiguration/Channel[2]/RealAxis/MechanicalElements/RotaryToLinearTransformation:
    ReferenceDistanceIsReadOnly = 1
    ReferenceDistance = 360
  DriveConfiguration/Channel[2]/RealAxis/Controller:
    ModeIsReadOnly = 1
    Mode = PositionControllerWithTorqueFeedForward
  DriveConfiguration/Channel[2]/RealAxis/Controller/Mode/Position:
    ProportionalGainIsReadOnly = 1
    ProportionalGain = 15.0
    IntegrationTimeIsReadOnly = 1
  DriveConfiguration/Channel[2]/RealAxis/Controller/Mode/Speed:
    ProportionalGainIsReadOnly = 1
    ProportionalGain = 8.0
    IntegrationTimeIsReadOnly = 1
    FilterTimeIsReadOnly = 1
  DriveConfiguration/Channel[2]/RealAxis/Controller/Mode:
    FeedForwardIsReadOnly = 1
    FeedForward = CyclicValueFromAxesGroup
  DriveConfiguration/Channel[2]/RealAxis/Controller/Mode/LoopFilters:
    LoopFilterXIsReadOnly = 1
  DriveConfiguration/Channel[2]/RealAxis/Homing:
    Mode = AbsoluteCorrection
    RestorePositionVariable = 
  DriveConfiguration/Channel[2]/RealAxis/StopReaction:
    DriveError = CyclicDecelerationFromAxesGroup
  DriveConfiguration/Channel[2]/RealAxis/MovementErrorLimits:
    PositionError = 0.5
  DriveConfiguration/Channel[2]/RealAxis:
    JerkFilterIsReadOnly = 1
    JerkFilter = Used
  DriveConfiguration/Channel[2]/RealAxis/JerkFilter:
    JerkTimeMin = 0.07
    JerkTime = 0.07
  DriveConfiguration/Channel[3]/RealAxis:
    AxisReference = gAxisQ3_D4r1100R_4
  DriveConfiguration/Channel[3]/RealAxis/MechanicalElements/Gearbox:
    InputIsReadOnly = 1
    Input = 77
    OutputIsReadOnly = 1
    Output = 2
  DriveConfiguration/Channel[3]/RealAxis/MechanicalElements/RotaryToLinearTransformation:
    ReferenceDistanceIsReadOnly = 1
    ReferenceDistance = 360
  DriveConfiguration/Channel[3]/RealAxis/Controller:
    ModeIsReadOnly = 1
    Mode = PositionControllerWithTorqueFeedForward
  DriveConfiguration/Channel[3]/RealAxis/Controller/Mode/Position:
    ProportionalGainIsReadOnly = 1
    ProportionalGain = 15.0
    IntegrationTimeIsReadOnly = 1
  DriveConfiguration/Channel[3]/RealAxis/Controller/Mode/Speed:
    ProportionalGainIsReadOnly = 1
    ProportionalGain = 8.0
    IntegrationTimeIsReadOnly = 1
    FilterTimeIsReadOnly = 1
  DriveConfiguration/Channel[3]/RealAxis/Controller/Mode:
    FeedForwardIsReadOnly = 1
    FeedForward = CyclicValueFromAxesGroup
  DriveConfiguration/Channel[3]/RealAxis/Controller/Mode/LoopFilters:
    LoopFilterXIsReadOnly = 1
  DriveConfiguration/Channel[3]/RealAxis/Homing:
    Mode = AbsoluteCorrection
    RestorePositionVariable = 
  DriveConfiguration/Channel[3]/RealAxis/StopReaction:
    DriveError = CyclicDecelerationFromAxesGroup
  DriveConfiguration/Channel[3]/RealAxis/MovementErrorLimits:
    PositionError = 0.5
  DriveConfiguration/Channel[3]/RealAxis:
    JerkFilterIsReadOnly = 1
    JerkFilter = Used
  DriveConfiguration/Channel[3]/RealAxis/JerkFilter:
    JerkTimeMin = 0.07
    JerkTime = 0.07
8EI8X8HWT10.xxxx-1-Q1-Q2-Q3_D4r1100R_5 : 8EI8X8HWT10.xxxx-1 v2.4.0.0 (NodeNumber=9)  [PLK1 -> 8EI2X2HWS10.xxxx-1-QC_D4r1100R_4.PLK2 [Cable Type=PowerlinkCable, Length=10, Version=1.0.0.3]; PLK2 -> 8EI2X2HWS10.xxxx-1-QC_D4r1100R_5.PLK1 [Cable Type=PowerlinkCable, Length=10, Version=1.0.0.3]; MT2 -> 8LSA46.DB060S200-3-Q2_D4r1100R_5.MT; MT3 -> 8LSA46.DB060S200-3-Q3_D4r1100R_5.MT]
  DriveConfiguration/Module:
    ActivateACOPOSSimulationOnPLC = 1
  DriveConfiguration/Encoder/EncoderX41:
    InterfaceType = EnDat
  DriveConfiguration/Encoder/EncoderX42:
    InterfaceType = EnDat
  DriveConfiguration/Encoder/EncoderX43:
    InterfaceType = EnDat
  DriveConfiguration/Channel[1]/RealAxis:
    AxisReference = gAxisQ1_D4r1100R_5
  DriveConfiguration/Channel[1]/RealAxis/MechanicalElements/Gearbox:
    InputIsReadOnly = 1
    Input = 77
    OutputIsReadOnly = 1
    Output = 2
  DriveConfiguration/Channel[1]/RealAxis/MechanicalElements/RotaryToLinearTransformation:
    ReferenceDistanceIsReadOnly = 1
    ReferenceDistance = 360
  DriveConfiguration/Channel[1]/RealAxis/Controller:
    ModeIsReadOnly = 1
    Mode = PositionControllerWithTorqueFeedForward
  DriveConfiguration/Channel[1]/RealAxis/Controller/Mode/Position:
    ProportionalGainIsReadOnly = 1
    ProportionalGain = 15.0
    IntegrationTimeIsReadOnly = 1
  DriveConfiguration/Channel[1]/RealAxis/Controller/Mode/Speed:
    ProportionalGainIsReadOnly = 1
    ProportionalGain = 8.0
    IntegrationTimeIsReadOnly = 1
    FilterTimeIsReadOnly = 1
  DriveConfiguration/Channel[1]/RealAxis/Controller/Mode:
    FeedForwardIsReadOnly = 1
    FeedForward = CyclicValueFromAxesGroup
  DriveConfiguration/Channel[1]/RealAxis/Controller/Mode/LoopFilters:
    LoopFilterXIsReadOnly = 1
  DriveConfiguration/Channel[1]/RealAxis/Homing:
    Mode = AbsoluteCorrection
    RestorePositionVariable = 
  DriveConfiguration/Channel[1]/RealAxis/StopReaction:
    DriveError = CyclicDecelerationFromAxesGroup
  DriveConfiguration/Channel[1]/RealAxis/MovementErrorLimits:
    PositionError = 0.5
  DriveConfiguration/Channel[1]/RealAxis:
    JerkFilterIsReadOnly = 1
    JerkFilter = Used
  DriveConfiguration/Channel[1]/RealAxis/JerkFilter:
    JerkTimeMin = 0.07
    JerkTime = 0.07
  DriveConfiguration/Channel[2]/RealAxis:
    AxisReference = gAxisQ2_D4r1100R_5
  DriveConfiguration/Channel[2]/RealAxis/MechanicalElements/Gearbox:
    InputIsReadOnly = 1
    Input = 77
    OutputIsReadOnly = 1
    Output = 2
  DriveConfiguration/Channel[2]/RealAxis/MechanicalElements/RotaryToLinearTransformation:
    ReferenceDistanceIsReadOnly = 1
    ReferenceDistance = 360
  DriveConfiguration/Channel[2]/RealAxis/Controller:
    ModeIsReadOnly = 1
    Mode = PositionControllerWithTorqueFeedForward
  DriveConfiguration/Channel[2]/RealAxis/Controller/Mode/Position:
    ProportionalGainIsReadOnly = 1
    ProportionalGain = 15.0
    IntegrationTimeIsReadOnly = 1
  DriveConfiguration/Channel[2]/RealAxis/Controller/Mode/Speed:
    ProportionalGainIsReadOnly = 1
    ProportionalGain = 8.0
    IntegrationTimeIsReadOnly = 1
    FilterTimeIsReadOnly = 1
  DriveConfiguration/Channel[2]/RealAxis/Controller/Mode:
    FeedForwardIsReadOnly = 1
    FeedForward = CyclicValueFromAxesGroup
  DriveConfiguration/Channel[2]/RealAxis/Controller/Mode/LoopFilters:
    LoopFilterXIsReadOnly = 1
  DriveConfiguration/Channel[2]/RealAxis/Homing:
    Mode = AbsoluteCorrection
    RestorePositionVariable = 
  DriveConfiguration/Channel[2]/RealAxis/StopReaction:
    DriveError = CyclicDecelerationFromAxesGroup
  DriveConfiguration/Channel[2]/RealAxis/MovementErrorLimits:
    PositionError = 0.5
  DriveConfiguration/Channel[2]/RealAxis:
    JerkFilterIsReadOnly = 1
    JerkFilter = Used
  DriveConfiguration/Channel[2]/RealAxis/JerkFilter:
    JerkTimeMin = 0.07
    JerkTime = 0.07
  DriveConfiguration/Channel[3]/RealAxis:
    AxisReference = gAxisQ3_D4r1100R_5
  DriveConfiguration/Channel[3]/RealAxis/MechanicalElements/Gearbox:
    InputIsReadOnly = 1
    Input = 77
    OutputIsReadOnly = 1
    Output = 2
  DriveConfiguration/Channel[3]/RealAxis/MechanicalElements/RotaryToLinearTransformation:
    ReferenceDistanceIsReadOnly = 1
    ReferenceDistance = 360
  DriveConfiguration/Channel[3]/RealAxis/Controller:
    ModeIsReadOnly = 1
    Mode = PositionControllerWithTorqueFeedForward
  DriveConfiguration/Channel[3]/RealAxis/Controller/Mode/Position:
    ProportionalGainIsReadOnly = 1
    ProportionalGain = 15.0
    IntegrationTimeIsReadOnly = 1
  DriveConfiguration/Channel[3]/RealAxis/Controller/Mode/Speed:
    ProportionalGainIsReadOnly = 1
    ProportionalGain = 8.0
    IntegrationTimeIsReadOnly = 1
    FilterTimeIsReadOnly = 1
  DriveConfiguration/Channel[3]/RealAxis/Controller/Mode:
    FeedForwardIsReadOnly = 1
    FeedForward = CyclicValueFromAxesGroup
  DriveConfiguration/Channel[3]/RealAxis/Controller/Mode/LoopFilters:
    LoopFilterXIsReadOnly = 1
  DriveConfiguration/Channel[3]/RealAxis/Homing:
    Mode = AbsoluteCorrection
    RestorePositionVariable = 
  DriveConfiguration/Channel[3]/RealAxis/StopReaction:
    DriveError = CyclicDecelerationFromAxesGroup
  DriveConfiguration/Channel[3]/RealAxis/MovementErrorLimits:
    PositionError = 0.5
  DriveConfiguration/Channel[3]/RealAxis:
    JerkFilterIsReadOnly = 1
    JerkFilter = Used
  DriveConfiguration/Channel[3]/RealAxis/JerkFilter:
    JerkTimeMin = 0.07
    JerkTime = 0.07
8EI8X8HWT10.xxxx-1-Q1-Q2-Q3_D4r1100R_6 : 8EI8X8HWT10.xxxx-1 v2.4.0.0 (NodeNumber=11)  [PLK1 -> 8EI2X2HWS10.xxxx-1-QC_D4r1100R_5.PLK2 [Cable Type=PowerlinkCable, Length=10, Version=1.0.0.3]; PLK2 -> 8EI2X2HWS10.xxxx-1-QC_D4r1100R_6.PLK1 [Cable Type=PowerlinkCable, Length=10, Version=1.0.0.3]; MT2 -> 8LSA46.DB060S200-3-Q2_D4r1100R_6.MT; MT3 -> 8LSA46.DB060S200-3-Q3_D4r1100R_6.MT]
  DriveConfiguration/Module:
    ActivateACOPOSSimulationOnPLC = 1
  DriveConfiguration/Encoder/EncoderX41:
    InterfaceType = EnDat
  DriveConfiguration/Encoder/EncoderX42:
    InterfaceType = EnDat
  DriveConfiguration/Encoder/EncoderX43:
    InterfaceType = EnDat
  DriveConfiguration/Channel[1]/RealAxis:
    AxisReference = gAxisQ1_D4r1100R_6
  DriveConfiguration/Channel[1]/RealAxis/MechanicalElements/Gearbox:
    InputIsReadOnly = 1
    Input = 77
    OutputIsReadOnly = 1
    Output = 2
  DriveConfiguration/Channel[1]/RealAxis/MechanicalElements/RotaryToLinearTransformation:
    ReferenceDistanceIsReadOnly = 1
    ReferenceDistance = 360
  DriveConfiguration/Channel[1]/RealAxis/Controller:
    ModeIsReadOnly = 1
    Mode = PositionControllerWithTorqueFeedForward
  DriveConfiguration/Channel[1]/RealAxis/Controller/Mode/Position:
    ProportionalGainIsReadOnly = 1
    ProportionalGain = 15.0
    IntegrationTimeIsReadOnly = 1
  DriveConfiguration/Channel[1]/RealAxis/Controller/Mode/Speed:
    ProportionalGainIsReadOnly = 1
    ProportionalGain = 8.0
    IntegrationTimeIsReadOnly = 1
    FilterTimeIsReadOnly = 1
  DriveConfiguration/Channel[1]/RealAxis/Controller/Mode:
    FeedForwardIsReadOnly = 1
    FeedForward = CyclicValueFromAxesGroup
  DriveConfiguration/Channel[1]/RealAxis/Controller/Mode/LoopFilters:
    LoopFilterXIsReadOnly = 1
  DriveConfiguration/Channel[1]/RealAxis/Homing:
    Mode = AbsoluteCorrection
    RestorePositionVariable = 
  DriveConfiguration/Channel[1]/RealAxis/StopReaction:
    DriveError = CyclicDecelerationFromAxesGroup
  DriveConfiguration/Channel[1]/RealAxis/MovementErrorLimits:
    PositionError = 0.5
  DriveConfiguration/Channel[1]/RealAxis:
    JerkFilterIsReadOnly = 1
    JerkFilter = Used
  DriveConfiguration/Channel[1]/RealAxis/JerkFilter:
    JerkTimeMin = 0.07
    JerkTime = 0.07
  DriveConfiguration/Channel[2]/RealAxis:
    AxisReference = gAxisQ2_D4r1100R_6
  DriveConfiguration/Channel[2]/RealAxis/MechanicalElements/Gearbox:
    InputIsReadOnly = 1
    Input = 77
    OutputIsReadOnly = 1
    Output = 2
  DriveConfiguration/Channel[2]/RealAxis/MechanicalElements/RotaryToLinearTransformation:
    ReferenceDistanceIsReadOnly = 1
    ReferenceDistance = 360
  DriveConfiguration/Channel[2]/RealAxis/Controller:
    ModeIsReadOnly = 1
    Mode = PositionControllerWithTorqueFeedForward
  DriveConfiguration/Channel[2]/RealAxis/Controller/Mode/Position:
    ProportionalGainIsReadOnly = 1
    ProportionalGain = 15.0
    IntegrationTimeIsReadOnly = 1
  DriveConfiguration/Channel[2]/RealAxis/Controller/Mode/Speed:
    ProportionalGainIsReadOnly = 1
    ProportionalGain = 8.0
    IntegrationTimeIsReadOnly = 1
    FilterTimeIsReadOnly = 1
  DriveConfiguration/Channel[2]/RealAxis/Controller/Mode:
    FeedForwardIsReadOnly = 1
    FeedForward = CyclicValueFromAxesGroup
  DriveConfiguration/Channel[2]/RealAxis/Controller/Mode/LoopFilters:
    LoopFilterXIsReadOnly = 1
  DriveConfiguration/Channel[2]/RealAxis/Homing:
    Mode = AbsoluteCorrection
    RestorePositionVariable = 
  DriveConfiguration/Channel[2]/RealAxis/StopReaction:
    DriveError = CyclicDecelerationFromAxesGroup
  DriveConfiguration/Channel[2]/RealAxis/MovementErrorLimits:
    PositionError = 0.5
  DriveConfiguration/Channel[2]/RealAxis:
    JerkFilterIsReadOnly = 1
    JerkFilter = Used
  DriveConfiguration/Channel[2]/RealAxis/JerkFilter:
    JerkTimeMin = 0.07
    JerkTime = 0.07
  DriveConfiguration/Channel[3]/RealAxis:
    AxisReference = gAxisQ3_D4r1100R_6
  DriveConfiguration/Channel[3]/RealAxis/MechanicalElements/Gearbox:
    InputIsReadOnly = 1
    Input = 77
    OutputIsReadOnly = 1
    Output = 2
  DriveConfiguration/Channel[3]/RealAxis/MechanicalElements/RotaryToLinearTransformation:
    ReferenceDistanceIsReadOnly = 1
    ReferenceDistance = 360
  DriveConfiguration/Channel[3]/RealAxis/Controller:
    ModeIsReadOnly = 1
    Mode = PositionControllerWithTorqueFeedForward
  DriveConfiguration/Channel[3]/RealAxis/Controller/Mode/Position:
    ProportionalGainIsReadOnly = 1
    ProportionalGain = 15.0
    IntegrationTimeIsReadOnly = 1
  DriveConfiguration/Channel[3]/RealAxis/Controller/Mode/Speed:
    ProportionalGainIsReadOnly = 1
    ProportionalGain = 8.0
    IntegrationTimeIsReadOnly = 1
    FilterTimeIsReadOnly = 1
  DriveConfiguration/Channel[3]/RealAxis/Controller/Mode:
    FeedForwardIsReadOnly = 1
    FeedForward = CyclicValueFromAxesGroup
  DriveConfiguration/Channel[3]/RealAxis/Controller/Mode/LoopFilters:
    LoopFilterXIsReadOnly = 1
  DriveConfiguration/Channel[3]/RealAxis/Homing:
    Mode = AbsoluteCorrection
    RestorePositionVariable = 
  DriveConfiguration/Channel[3]/RealAxis/StopReaction:
    DriveError = CyclicDecelerationFromAxesGroup
  DriveConfiguration/Channel[3]/RealAxis/MovementErrorLimits:
    PositionError = 0.5
  DriveConfiguration/Channel[3]/RealAxis:
    JerkFilterIsReadOnly = 1
    JerkFilter = Used
  DriveConfiguration/Channel[3]/RealAxis/JerkFilter:
    JerkTimeMin = 0.07
    JerkTime = 0.07
8LSA25.D9060S000-3 : 8LSA25.D9060S000-3 v2.2.0.2  [MT -> 8EI2X2HWT10.xxxx-1.MT3]
  M1/MotorParameters:
    MOTOR_AMB_TEMP_RATED = 40
  M1/MotorParameters/TemperatureSensor:
    MOTOR_TEMPSENS_LIM = 130
8LSA25.D9060S000-3_a : 8LSA25.D9060S000-3 v2.2.0.2  [MT -> 8EI2X2HWT10.xxxx-1.MT1]
  M1/MotorParameters:
    MOTOR_AMB_TEMP_RATED = 40
  M1/MotorParameters/TemperatureSensor:
    MOTOR_TEMPSENS_LIM = 130
8LSA25.D9060S000-3_b : 8LSA25.D9060S000-3 v2.2.0.2  [MT -> 8EI2X2HWT10.xxxx-1.MT2]
  M1/MotorParameters:
    MOTOR_AMB_TEMP_RATED = 40
  M1/MotorParameters/TemperatureSensor:
    MOTOR_TEMPSENS_LIM = 130
8LSA35.DB030S200-3-QC_D4r1100R_1 : MotorSynchronous_any v2.2.1.0  [MT -> 8EI2X2HWS10.xxxx-1-QC_D4r1100R_1.MT1]
  M1/MotorParameters:
    MOTOR_POLEPAIRS = 4
    MOTOR_SPEED_RATED = 3000
    MOTOR_SPEED_MAX = 9000
    MOTOR_VOLTAGE_RATED = 400
    MOTOR_CURR_RATED = 1.4
    MOTOR_CURR_STALL = 1.6
    MOTOR_CURR_MAX = 6.8
    MOTOR_TORQ_RATED = 2.1
    MOTOR_TORQ_STALL = 2.3
    MOTOR_TORQ_MAX = 9.2
    MOTOR_VOLTAGE_CONST = 87.96
    MOTOR_TORQ_CONST = 1.45
    MOTOR_STATOR_RESISTANCE = 12.22
    MOTOR_STATOR_INDUCTANCE = 63
    MOTOR_INERTIA = 0.9
    VoltageLimitation = Used
  M1/MotorParameters/VoltageLimitation:
    MOTOR_UDC_MAX = 1000
  M1/MotorParameters/EncoderMounting:
    Angle = StoredOnEncoder
  M1/MotorParameters/TemperatureSensor:
    MOTOR_TEMPSENS_LIM = 130
    TemperatureSensorInterface = EncoderConnectorDigital
    MOTOR_TEMPSENS_PAR1 = 30
    MOTOR_TEMPSENS_PAR2 = 254
    MOTOR_TEMPSENS_PAR3 = -29.72
    MOTOR_TEMPSENS_PAR4 = -4.58
    MOTOR_TEMPSENS_PAR5 = 20.33
    MOTOR_TEMPSENS_PAR6 = 45.18
    MOTOR_TEMPSENS_PAR7 = 69.96
    MOTOR_TEMPSENS_PAR8 = 94.71
    MOTOR_TEMPSENS_PAR9 = 119.6
    MOTOR_TEMPSENS_PAR10 = 149.11
  M1/MotorParameters/TemperatureModel:
    MOTOR_WIND_TEMP_MAX = 110
  M1/MotorParameters/TemperatureModel/Calculation:
    MOTOR_WIND_CROSS_SECT = 0.181
    MOTOR_TAU_THERM = 2040
  M1:
    Brake = Used
  M1/Brake:
    MOTOR_BRAKE_CURR_RATED = 0.56
    MOTOR_BRAKE_TORQ_RATED = 4
    MOTOR_BRAKE_ON_TIME = 0.01
    MOTOR_BRAKE_OFF_TIME = 0.06
    MOTOR_BRAKE_INERTIA = 0.38
  M1/Encoder:
    MOTOR_ENCOD_ATTR = 1
    MOTOR_ENCOD_INERTIA = 0.022
    TemperatureSensor = Used
  M1/Encoder/TemperatureSensor:
    MOTOR_ENCOD_TEMP_LIM = 129
  M1:
    Gearbox = UsedWithDynamicTorqueLimitation
  M1/Gearbox/GearRatio:
    Input = 10
  M1/Gearbox:
    MOTORGEAR_SPEED_MAX = 7500
    MOTORGEAR_TORQ_NOM = 24.0
    MOTORGEAR_TORQ_MAX = 24.0
    MOTORGEAR_INERTIA = 0.16
    MOTORGEAR_VISC_FRIC = 0.001
    MOTORGEAR_STAT_FRIC = 0.1
8LSA35.DB030S200-3-QC_D4r1100R_2 : MotorSynchronous_any v2.2.1.0  [MT -> 8EI2X2HWS10.xxxx-1-QC_D4r1100R_2.MT1]
  M1/MotorParameters:
    MOTOR_POLEPAIRS = 4
    MOTOR_SPEED_RATED = 3000
    MOTOR_SPEED_MAX = 9000
    MOTOR_VOLTAGE_RATED = 400
    MOTOR_CURR_RATED = 1.4
    MOTOR_CURR_STALL = 1.6
    MOTOR_CURR_MAX = 6.8
    MOTOR_TORQ_RATED = 2.1
    MOTOR_TORQ_STALL = 2.3
    MOTOR_TORQ_MAX = 9.2
    MOTOR_VOLTAGE_CONST = 87.96
    MOTOR_TORQ_CONST = 1.45
    MOTOR_STATOR_RESISTANCE = 12.22
    MOTOR_STATOR_INDUCTANCE = 63
    MOTOR_INERTIA = 0.9
    VoltageLimitation = Used
  M1/MotorParameters/VoltageLimitation:
    MOTOR_UDC_MAX = 1000
  M1/MotorParameters/EncoderMounting:
    Angle = StoredOnEncoder
  M1/MotorParameters/TemperatureSensor:
    MOTOR_TEMPSENS_LIM = 130
    TemperatureSensorInterface = EncoderConnectorDigital
    MOTOR_TEMPSENS_PAR1 = 30
    MOTOR_TEMPSENS_PAR2 = 254
    MOTOR_TEMPSENS_PAR3 = -29.72
    MOTOR_TEMPSENS_PAR4 = -4.58
    MOTOR_TEMPSENS_PAR5 = 20.33
    MOTOR_TEMPSENS_PAR6 = 45.18
    MOTOR_TEMPSENS_PAR7 = 69.96
    MOTOR_TEMPSENS_PAR8 = 94.71
    MOTOR_TEMPSENS_PAR9 = 119.6
    MOTOR_TEMPSENS_PAR10 = 149.11
  M1/MotorParameters/TemperatureModel:
    MOTOR_WIND_TEMP_MAX = 110
  M1/MotorParameters/TemperatureModel/Calculation:
    MOTOR_WIND_CROSS_SECT = 0.181
    MOTOR_TAU_THERM = 2040
  M1:
    Brake = Used
  M1/Brake:
    MOTOR_BRAKE_CURR_RATED = 0.56
    MOTOR_BRAKE_TORQ_RATED = 4
    MOTOR_BRAKE_ON_TIME = 0.01
    MOTOR_BRAKE_OFF_TIME = 0.06
    MOTOR_BRAKE_INERTIA = 0.38
  M1/Encoder:
    MOTOR_ENCOD_ATTR = 1
    MOTOR_ENCOD_INERTIA = 0.022
    TemperatureSensor = Used
  M1/Encoder/TemperatureSensor:
    MOTOR_ENCOD_TEMP_LIM = 129
  M1:
    Gearbox = UsedWithDynamicTorqueLimitation
  M1/Gearbox/GearRatio:
    Input = 10
  M1/Gearbox:
    MOTORGEAR_SPEED_MAX = 7500
    MOTORGEAR_TORQ_NOM = 24.0
    MOTORGEAR_TORQ_MAX = 24.0
    MOTORGEAR_INERTIA = 0.16
    MOTORGEAR_VISC_FRIC = 0.001
    MOTORGEAR_STAT_FRIC = 0.1
8LSA35.DB030S200-3-QC_D4r1100R_3 : MotorSynchronous_any v2.2.1.0  [MT -> 8EI2X2HWS10.xxxx-1-QC_D4r1100R_3.MT1]
  M1/MotorParameters:
    MOTOR_POLEPAIRS = 4
    MOTOR_SPEED_RATED = 3000
    MOTOR_SPEED_MAX = 9000
    MOTOR_VOLTAGE_RATED = 400
    MOTOR_CURR_RATED = 1.4
    MOTOR_CURR_STALL = 1.6
    MOTOR_CURR_MAX = 6.8
    MOTOR_TORQ_RATED = 2.1
    MOTOR_TORQ_STALL = 2.3
    MOTOR_TORQ_MAX = 9.2
    MOTOR_VOLTAGE_CONST = 87.96
    MOTOR_TORQ_CONST = 1.45
    MOTOR_STATOR_RESISTANCE = 12.22
    MOTOR_STATOR_INDUCTANCE = 63
    MOTOR_INERTIA = 0.9
    VoltageLimitation = Used
  M1/MotorParameters/VoltageLimitation:
    MOTOR_UDC_MAX = 1000
  M1/MotorParameters/EncoderMounting:
    Angle = StoredOnEncoder
  M1/MotorParameters/TemperatureSensor:
    MOTOR_TEMPSENS_LIM = 130
    TemperatureSensorInterface = EncoderConnectorDigital
    MOTOR_TEMPSENS_PAR1 = 30
    MOTOR_TEMPSENS_PAR2 = 254
    MOTOR_TEMPSENS_PAR3 = -29.72
    MOTOR_TEMPSENS_PAR4 = -4.58
    MOTOR_TEMPSENS_PAR5 = 20.33
    MOTOR_TEMPSENS_PAR6 = 45.18
    MOTOR_TEMPSENS_PAR7 = 69.96
    MOTOR_TEMPSENS_PAR8 = 94.71
    MOTOR_TEMPSENS_PAR9 = 119.6
    MOTOR_TEMPSENS_PAR10 = 149.11
  M1/MotorParameters/TemperatureModel:
    MOTOR_WIND_TEMP_MAX = 110
  M1/MotorParameters/TemperatureModel/Calculation:
    MOTOR_WIND_CROSS_SECT = 0.181
    MOTOR_TAU_THERM = 2040
  M1:
    Brake = Used
  M1/Brake:
    MOTOR_BRAKE_CURR_RATED = 0.56
    MOTOR_BRAKE_TORQ_RATED = 4
    MOTOR_BRAKE_ON_TIME = 0.01
    MOTOR_BRAKE_OFF_TIME = 0.06
    MOTOR_BRAKE_INERTIA = 0.38
  M1/Encoder:
    MOTOR_ENCOD_ATTR = 1
    MOTOR_ENCOD_INERTIA = 0.022
    TemperatureSensor = Used
  M1/Encoder/TemperatureSensor:
    MOTOR_ENCOD_TEMP_LIM = 129
  M1:
    Gearbox = UsedWithDynamicTorqueLimitation
  M1/Gearbox/GearRatio:
    Input = 10
  M1/Gearbox:
    MOTORGEAR_SPEED_MAX = 7500
    MOTORGEAR_TORQ_NOM = 24.0
    MOTORGEAR_TORQ_MAX = 24.0
    MOTORGEAR_INERTIA = 0.16
    MOTORGEAR_VISC_FRIC = 0.001
    MOTORGEAR_STAT_FRIC = 0.1
8LSA35.DB030S200-3-QC_D4r1100R_4 : MotorSynchronous_any v2.2.1.0  [MT -> 8EI2X2HWS10.xxxx-1-QC_D4r1100R_4.MT1]
  M1/MotorParameters:
    MOTOR_POLEPAIRS = 4
    MOTOR_SPEED_RATED = 3000
    MOTOR_SPEED_MAX = 9000
    MOTOR_VOLTAGE_RATED = 400
    MOTOR_CURR_RATED = 1.4
    MOTOR_CURR_STALL = 1.6
    MOTOR_CURR_MAX = 6.8
    MOTOR_TORQ_RATED = 2.1
    MOTOR_TORQ_STALL = 2.3
    MOTOR_TORQ_MAX = 9.2
    MOTOR_VOLTAGE_CONST = 87.96
    MOTOR_TORQ_CONST = 1.45
    MOTOR_STATOR_RESISTANCE = 12.22
    MOTOR_STATOR_INDUCTANCE = 63
    MOTOR_INERTIA = 0.9
    VoltageLimitation = Used
  M1/MotorParameters/VoltageLimitation:
    MOTOR_UDC_MAX = 1000
  M1/MotorParameters/EncoderMounting:
    Angle = StoredOnEncoder
  M1/MotorParameters/TemperatureSensor:
    MOTOR_TEMPSENS_LIM = 130
    TemperatureSensorInterface = EncoderConnectorDigital
    MOTOR_TEMPSENS_PAR1 = 30
    MOTOR_TEMPSENS_PAR2 = 254
    MOTOR_TEMPSENS_PAR3 = -29.72
    MOTOR_TEMPSENS_PAR4 = -4.58
    MOTOR_TEMPSENS_PAR5 = 20.33
    MOTOR_TEMPSENS_PAR6 = 45.18
    MOTOR_TEMPSENS_PAR7 = 69.96
    MOTOR_TEMPSENS_PAR8 = 94.71
    MOTOR_TEMPSENS_PAR9 = 119.6
    MOTOR_TEMPSENS_PAR10 = 149.11
  M1/MotorParameters/TemperatureModel:
    MOTOR_WIND_TEMP_MAX = 110
  M1/MotorParameters/TemperatureModel/Calculation:
    MOTOR_WIND_CROSS_SECT = 0.181
    MOTOR_TAU_THERM = 2040
  M1:
    Brake = Used
  M1/Brake:
    MOTOR_BRAKE_CURR_RATED = 0.56
    MOTOR_BRAKE_TORQ_RATED = 4
    MOTOR_BRAKE_ON_TIME = 0.01
    MOTOR_BRAKE_OFF_TIME = 0.06
    MOTOR_BRAKE_INERTIA = 0.38
  M1/Encoder:
    MOTOR_ENCOD_ATTR = 1
    MOTOR_ENCOD_INERTIA = 0.022
    TemperatureSensor = Used
  M1/Encoder/TemperatureSensor:
    MOTOR_ENCOD_TEMP_LIM = 129
  M1:
    Gearbox = UsedWithDynamicTorqueLimitation
  M1/Gearbox/GearRatio:
    Input = 10
  M1/Gearbox:
    MOTORGEAR_SPEED_MAX = 7500
    MOTORGEAR_TORQ_NOM = 24.0
    MOTORGEAR_TORQ_MAX = 24.0
    MOTORGEAR_INERTIA = 0.16
    MOTORGEAR_VISC_FRIC = 0.001
    MOTORGEAR_STAT_FRIC = 0.1
8LSA35.DB030S200-3-QC_D4r1100R_5 : MotorSynchronous_any v2.2.1.0  [MT -> 8EI2X2HWS10.xxxx-1-QC_D4r1100R_5.MT1]
  M1/MotorParameters:
    MOTOR_POLEPAIRS = 4
    MOTOR_SPEED_RATED = 3000
    MOTOR_SPEED_MAX = 9000
    MOTOR_VOLTAGE_RATED = 400
    MOTOR_CURR_RATED = 1.4
    MOTOR_CURR_STALL = 1.6
    MOTOR_CURR_MAX = 6.8
    MOTOR_TORQ_RATED = 2.1
    MOTOR_TORQ_STALL = 2.3
    MOTOR_TORQ_MAX = 9.2
    MOTOR_VOLTAGE_CONST = 87.96
    MOTOR_TORQ_CONST = 1.45
    MOTOR_STATOR_RESISTANCE = 12.22
    MOTOR_STATOR_INDUCTANCE = 63
    MOTOR_INERTIA = 0.9
    VoltageLimitation = Used
  M1/MotorParameters/VoltageLimitation:
    MOTOR_UDC_MAX = 1000
  M1/MotorParameters/EncoderMounting:
    Angle = StoredOnEncoder
  M1/MotorParameters/TemperatureSensor:
    MOTOR_TEMPSENS_LIM = 130
    TemperatureSensorInterface = EncoderConnectorDigital
    MOTOR_TEMPSENS_PAR1 = 30
    MOTOR_TEMPSENS_PAR2 = 254
    MOTOR_TEMPSENS_PAR3 = -29.72
    MOTOR_TEMPSENS_PAR4 = -4.58
    MOTOR_TEMPSENS_PAR5 = 20.33
    MOTOR_TEMPSENS_PAR6 = 45.18
    MOTOR_TEMPSENS_PAR7 = 69.96
    MOTOR_TEMPSENS_PAR8 = 94.71
    MOTOR_TEMPSENS_PAR9 = 119.6
    MOTOR_TEMPSENS_PAR10 = 149.11
  M1/MotorParameters/TemperatureModel:
    MOTOR_WIND_TEMP_MAX = 110
  M1/MotorParameters/TemperatureModel/Calculation:
    MOTOR_WIND_CROSS_SECT = 0.181
    MOTOR_TAU_THERM = 2040
  M1:
    Brake = Used
  M1/Brake:
    MOTOR_BRAKE_CURR_RATED = 0.56
    MOTOR_BRAKE_TORQ_RATED = 4
    MOTOR_BRAKE_ON_TIME = 0.01
    MOTOR_BRAKE_OFF_TIME = 0.06
    MOTOR_BRAKE_INERTIA = 0.38
  M1/Encoder:
    MOTOR_ENCOD_ATTR = 1
    MOTOR_ENCOD_INERTIA = 0.022
    TemperatureSensor = Used
  M1/Encoder/TemperatureSensor:
    MOTOR_ENCOD_TEMP_LIM = 129
  M1:
    Gearbox = UsedWithDynamicTorqueLimitation
  M1/Gearbox/GearRatio:
    Input = 10
  M1/Gearbox:
    MOTORGEAR_SPEED_MAX = 7500
    MOTORGEAR_TORQ_NOM = 24.0
    MOTORGEAR_TORQ_MAX = 24.0
    MOTORGEAR_INERTIA = 0.16
    MOTORGEAR_VISC_FRIC = 0.001
    MOTORGEAR_STAT_FRIC = 0.1
8LSA35.DB030S200-3-QC_D4r1100R_6 : MotorSynchronous_any v2.2.1.0  [MT -> 8EI2X2HWS10.xxxx-1-QC_D4r1100R_6.MT1]
  M1/MotorParameters:
    MOTOR_POLEPAIRS = 4
    MOTOR_SPEED_RATED = 3000
    MOTOR_SPEED_MAX = 9000
    MOTOR_VOLTAGE_RATED = 400
    MOTOR_CURR_RATED = 1.4
    MOTOR_CURR_STALL = 1.6
    MOTOR_CURR_MAX = 6.8
    MOTOR_TORQ_RATED = 2.1
    MOTOR_TORQ_STALL = 2.3
    MOTOR_TORQ_MAX = 9.2
    MOTOR_VOLTAGE_CONST = 87.96
    MOTOR_TORQ_CONST = 1.45
    MOTOR_STATOR_RESISTANCE = 12.22
    MOTOR_STATOR_INDUCTANCE = 63
    MOTOR_INERTIA = 0.9
    VoltageLimitation = Used
  M1/MotorParameters/VoltageLimitation:
    MOTOR_UDC_MAX = 1000
  M1/MotorParameters/EncoderMounting:
    Angle = StoredOnEncoder
  M1/MotorParameters/TemperatureSensor:
    MOTOR_TEMPSENS_LIM = 130
    TemperatureSensorInterface = EncoderConnectorDigital
    MOTOR_TEMPSENS_PAR1 = 30
    MOTOR_TEMPSENS_PAR2 = 254
    MOTOR_TEMPSENS_PAR3 = -29.72
    MOTOR_TEMPSENS_PAR4 = -4.58
    MOTOR_TEMPSENS_PAR5 = 20.33
    MOTOR_TEMPSENS_PAR6 = 45.18
    MOTOR_TEMPSENS_PAR7 = 69.96
    MOTOR_TEMPSENS_PAR8 = 94.71
    MOTOR_TEMPSENS_PAR9 = 119.6
    MOTOR_TEMPSENS_PAR10 = 149.11
  M1/MotorParameters/TemperatureModel:
    MOTOR_WIND_TEMP_MAX = 110
  M1/MotorParameters/TemperatureModel/Calculation:
    MOTOR_WIND_CROSS_SECT = 0.181
    MOTOR_TAU_THERM = 2040
  M1:
    Brake = Used
  M1/Brake:
    MOTOR_BRAKE_CURR_RATED = 0.56
    MOTOR_BRAKE_TORQ_RATED = 4
    MOTOR_BRAKE_ON_TIME = 0.01
    MOTOR_BRAKE_OFF_TIME = 0.06
    MOTOR_BRAKE_INERTIA = 0.38
  M1/Encoder:
    MOTOR_ENCOD_ATTR = 1
    MOTOR_ENCOD_INERTIA = 0.022
    TemperatureSensor = Used
  M1/Encoder/TemperatureSensor:
    MOTOR_ENCOD_TEMP_LIM = 129
  M1:
    Gearbox = UsedWithDynamicTorqueLimitation
  M1/Gearbox/GearRatio:
    Input = 10
  M1/Gearbox:
    MOTORGEAR_SPEED_MAX = 7500
    MOTORGEAR_TORQ_NOM = 24.0
    MOTORGEAR_TORQ_MAX = 24.0
    MOTORGEAR_INERTIA = 0.16
    MOTORGEAR_VISC_FRIC = 0.001
    MOTORGEAR_STAT_FRIC = 0.1
8LSA46.DB060S200-3-Q1_D4r1100R_1 : MotorSynchronous_any v2.2.1.0  [MT -> 8EI8X8HWT10.xxxx-1-Q1-Q2-Q3_D4r1100R_1.MT1]
  M1/MotorParameters:
    MOTOR_POLEPAIRS = 5
    MOTOR_SPEED_RATED = 6000
    MOTOR_SPEED_MAX = 12000
    MOTOR_VOLTAGE_RATED = 400
    MOTOR_CURR_RATED = 6.1
    MOTOR_CURR_STALL = 12.3
    MOTOR_CURR_MAX = 72.9
    MOTOR_TORQ_RATED = 5
    MOTOR_TORQ_STALL = 10
    MOTOR_TORQ_MAX = 38
    MOTOR_VOLTAGE_CONST = 49.22
    MOTOR_TORQ_CONST = 0.81
    MOTOR_STATOR_RESISTANCE = 0.48
    MOTOR_STATOR_INDUCTANCE = 4.35938
    MOTOR_INERTIA = 4.387
    VoltageLimitation = Used
  M1/MotorParameters/VoltageLimitation:
    MOTOR_UDC_MAX = 1000
  M1/MotorParameters/EncoderMounting:
    Angle = StoredOnEncoder
  M1/MotorParameters/TemperatureSensor:
    MOTOR_TEMPSENS_LIM = 130
    TemperatureSensorInterface = EncoderConnectorDigital
    MOTOR_TEMPSENS_PAR1 = 30
    MOTOR_TEMPSENS_PAR2 = 254
    MOTOR_TEMPSENS_PAR3 = -29.72
    MOTOR_TEMPSENS_PAR4 = -4.58
    MOTOR_TEMPSENS_PAR5 = 20.33
    MOTOR_TEMPSENS_PAR6 = 45.18
    MOTOR_TEMPSENS_PAR7 = 69.96
    MOTOR_TEMPSENS_PAR8 = 94.71
    MOTOR_TEMPSENS_PAR9 = 119.6
    MOTOR_TEMPSENS_PAR10 = 149.11
  M1/MotorParameters/TemperatureModel:
    MOTOR_WIND_TEMP_MAX = 110
  M1/MotorParameters/TemperatureModel/Calculation:
    MOTOR_WIND_CROSS_SECT = 1.765
    MOTOR_TAU_THERM = 2400
  M1:
    Brake = Used
  M1/Brake:
    MOTOR_BRAKE_CURR_RATED = 0.83
    MOTOR_BRAKE_TORQ_RATED = 8
    MOTOR_BRAKE_ON_TIME = 0.038
    MOTOR_BRAKE_OFF_TIME = 0.055
    MOTOR_BRAKE_INERTIA = 0.69
  M1/Encoder:
    MOTOR_ENCOD_ATTR = 1
    MOTOR_ENCOD_INERTIA = 0.026
    TemperatureSensor = Used
  M1/Encoder/TemperatureSensor:
    MOTOR_ENCOD_TEMP_LIM = 129
  M1:
    Gearbox = UsedWithDynamicTorqueLimitation
  M1/Gearbox/GearRatio:
    Input = 77
    Output = 2
  M1/Gearbox:
    MOTORGEAR_SPEED_MAX = 7500
    MOTORGEAR_TORQ_NOM = 424
    MOTORGEAR_TORQ_MAX = 424
    MOTORGEAR_INERTIA = 0.6
    MOTORGEAR_VISC_FRIC = 0.01
    MOTORGEAR_STAT_FRIC = 0.11
8LSA46.DB060S200-3-Q1_D4r1100R_2 : MotorSynchronous_any v2.2.1.0  [MT -> 8EI8X8HWT10.xxxx-1-Q1-Q2-Q3_D4r1100R_2.MT1]
  M1/MotorParameters:
    MOTOR_POLEPAIRS = 5
    MOTOR_SPEED_RATED = 6000
    MOTOR_SPEED_MAX = 12000
    MOTOR_VOLTAGE_RATED = 400
    MOTOR_CURR_RATED = 6.1
    MOTOR_CURR_STALL = 12.3
    MOTOR_CURR_MAX = 72.9
    MOTOR_TORQ_RATED = 5
    MOTOR_TORQ_STALL = 10
    MOTOR_TORQ_MAX = 38
    MOTOR_VOLTAGE_CONST = 49.22
    MOTOR_TORQ_CONST = 0.81
    MOTOR_STATOR_RESISTANCE = 0.48
    MOTOR_STATOR_INDUCTANCE = 4.35938
    MOTOR_INERTIA = 4.387
    VoltageLimitation = Used
  M1/MotorParameters/VoltageLimitation:
    MOTOR_UDC_MAX = 1000
  M1/MotorParameters/EncoderMounting:
    Angle = StoredOnEncoder
  M1/MotorParameters/TemperatureSensor:
    MOTOR_TEMPSENS_LIM = 130
    TemperatureSensorInterface = EncoderConnectorDigital
    MOTOR_TEMPSENS_PAR1 = 30
    MOTOR_TEMPSENS_PAR2 = 254
    MOTOR_TEMPSENS_PAR3 = -29.72
    MOTOR_TEMPSENS_PAR4 = -4.58
    MOTOR_TEMPSENS_PAR5 = 20.33
    MOTOR_TEMPSENS_PAR6 = 45.18
    MOTOR_TEMPSENS_PAR7 = 69.96
    MOTOR_TEMPSENS_PAR8 = 94.71
    MOTOR_TEMPSENS_PAR9 = 119.6
    MOTOR_TEMPSENS_PAR10 = 149.11
  M1/MotorParameters/TemperatureModel:
    MOTOR_WIND_TEMP_MAX = 110
  M1/MotorParameters/TemperatureModel/Calculation:
    MOTOR_WIND_CROSS_SECT = 1.765
    MOTOR_TAU_THERM = 2400
  M1:
    Brake = Used
  M1/Brake:
    MOTOR_BRAKE_CURR_RATED = 0.83
    MOTOR_BRAKE_TORQ_RATED = 8
    MOTOR_BRAKE_ON_TIME = 0.038
    MOTOR_BRAKE_OFF_TIME = 0.055
    MOTOR_BRAKE_INERTIA = 0.69
  M1/Encoder:
    MOTOR_ENCOD_ATTR = 1
    MOTOR_ENCOD_INERTIA = 0.026
    TemperatureSensor = Used
  M1/Encoder/TemperatureSensor:
    MOTOR_ENCOD_TEMP_LIM = 129
  M1:
    Gearbox = UsedWithDynamicTorqueLimitation
  M1/Gearbox/GearRatio:
    Input = 77
    Output = 2
  M1/Gearbox:
    MOTORGEAR_SPEED_MAX = 7500
    MOTORGEAR_TORQ_NOM = 424
    MOTORGEAR_TORQ_MAX = 424
    MOTORGEAR_INERTIA = 0.6
    MOTORGEAR_VISC_FRIC = 0.01
    MOTORGEAR_STAT_FRIC = 0.11
8LSA46.DB060S200-3-Q1_D4r1100R_3 : MotorSynchronous_any v2.2.1.0  [MT -> 8EI8X8HWT10.xxxx-1-Q1-Q2-Q3_D4r1100R_3.MT1]
  M1/MotorParameters:
    MOTOR_POLEPAIRS = 5
    MOTOR_SPEED_RATED = 6000
    MOTOR_SPEED_MAX = 12000
    MOTOR_VOLTAGE_RATED = 400
    MOTOR_CURR_RATED = 6.1
    MOTOR_CURR_STALL = 12.3
    MOTOR_CURR_MAX = 72.9
    MOTOR_TORQ_RATED = 5
    MOTOR_TORQ_STALL = 10
    MOTOR_TORQ_MAX = 38
    MOTOR_VOLTAGE_CONST = 49.22
    MOTOR_TORQ_CONST = 0.81
    MOTOR_STATOR_RESISTANCE = 0.48
    MOTOR_STATOR_INDUCTANCE = 4.35938
    MOTOR_INERTIA = 4.387
    VoltageLimitation = Used
  M1/MotorParameters/VoltageLimitation:
    MOTOR_UDC_MAX = 1000
  M1/MotorParameters/EncoderMounting:
    Angle = StoredOnEncoder
  M1/MotorParameters/TemperatureSensor:
    MOTOR_TEMPSENS_LIM = 130
    TemperatureSensorInterface = EncoderConnectorDigital
    MOTOR_TEMPSENS_PAR1 = 30
    MOTOR_TEMPSENS_PAR2 = 254
    MOTOR_TEMPSENS_PAR3 = -29.72
    MOTOR_TEMPSENS_PAR4 = -4.58
    MOTOR_TEMPSENS_PAR5 = 20.33
    MOTOR_TEMPSENS_PAR6 = 45.18
    MOTOR_TEMPSENS_PAR7 = 69.96
    MOTOR_TEMPSENS_PAR8 = 94.71
    MOTOR_TEMPSENS_PAR9 = 119.6
    MOTOR_TEMPSENS_PAR10 = 149.11
  M1/MotorParameters/TemperatureModel:
    MOTOR_WIND_TEMP_MAX = 110
  M1/MotorParameters/TemperatureModel/Calculation:
    MOTOR_WIND_CROSS_SECT = 1.765
    MOTOR_TAU_THERM = 2400
  M1:
    Brake = Used
  M1/Brake:
    MOTOR_BRAKE_CURR_RATED = 0.83
    MOTOR_BRAKE_TORQ_RATED = 8
    MOTOR_BRAKE_ON_TIME = 0.038
    MOTOR_BRAKE_OFF_TIME = 0.055
    MOTOR_BRAKE_INERTIA = 0.69
  M1/Encoder:
    MOTOR_ENCOD_ATTR = 1
    MOTOR_ENCOD_INERTIA = 0.026
    TemperatureSensor = Used
  M1/Encoder/TemperatureSensor:
    MOTOR_ENCOD_TEMP_LIM = 129
  M1:
    Gearbox = UsedWithDynamicTorqueLimitation
  M1/Gearbox/GearRatio:
    Input = 77
    Output = 2
  M1/Gearbox:
    MOTORGEAR_SPEED_MAX = 7500
    MOTORGEAR_TORQ_NOM = 424
    MOTORGEAR_TORQ_MAX = 424
    MOTORGEAR_INERTIA = 0.6
    MOTORGEAR_VISC_FRIC = 0.01
    MOTORGEAR_STAT_FRIC = 0.11
8LSA46.DB060S200-3-Q1_D4r1100R_4 : MotorSynchronous_any v2.2.1.0  [MT -> 8EI8X8HWT10.xxxx-1-Q1-Q2-Q3_D4r1100R_4.MT1]
  M1/MotorParameters:
    MOTOR_POLEPAIRS = 5
    MOTOR_SPEED_RATED = 6000
    MOTOR_SPEED_MAX = 12000
    MOTOR_VOLTAGE_RATED = 400
    MOTOR_CURR_RATED = 6.1
    MOTOR_CURR_STALL = 12.3
    MOTOR_CURR_MAX = 72.9
    MOTOR_TORQ_RATED = 5
    MOTOR_TORQ_STALL = 10
    MOTOR_TORQ_MAX = 38
    MOTOR_VOLTAGE_CONST = 49.22
    MOTOR_TORQ_CONST = 0.81
    MOTOR_STATOR_RESISTANCE = 0.48
    MOTOR_STATOR_INDUCTANCE = 4.35938
    MOTOR_INERTIA = 4.387
    VoltageLimitation = Used
  M1/MotorParameters/VoltageLimitation:
    MOTOR_UDC_MAX = 1000
  M1/MotorParameters/EncoderMounting:
    Angle = StoredOnEncoder
  M1/MotorParameters/TemperatureSensor:
    MOTOR_TEMPSENS_LIM = 130
    TemperatureSensorInterface = EncoderConnectorDigital
    MOTOR_TEMPSENS_PAR1 = 30
    MOTOR_TEMPSENS_PAR2 = 254
    MOTOR_TEMPSENS_PAR3 = -29.72
    MOTOR_TEMPSENS_PAR4 = -4.58
    MOTOR_TEMPSENS_PAR5 = 20.33
    MOTOR_TEMPSENS_PAR6 = 45.18
    MOTOR_TEMPSENS_PAR7 = 69.96
    MOTOR_TEMPSENS_PAR8 = 94.71
    MOTOR_TEMPSENS_PAR9 = 119.6
    MOTOR_TEMPSENS_PAR10 = 149.11
  M1/MotorParameters/TemperatureModel:
    MOTOR_WIND_TEMP_MAX = 110
  M1/MotorParameters/TemperatureModel/Calculation:
    MOTOR_WIND_CROSS_SECT = 1.765
    MOTOR_TAU_THERM = 2400
  M1:
    Brake = Used
  M1/Brake:
    MOTOR_BRAKE_CURR_RATED = 0.83
    MOTOR_BRAKE_TORQ_RATED = 8
    MOTOR_BRAKE_ON_TIME = 0.038
    MOTOR_BRAKE_OFF_TIME = 0.055
    MOTOR_BRAKE_INERTIA = 0.69
  M1/Encoder:
    MOTOR_ENCOD_ATTR = 1
    MOTOR_ENCOD_INERTIA = 0.026
    TemperatureSensor = Used
  M1/Encoder/TemperatureSensor:
    MOTOR_ENCOD_TEMP_LIM = 129
  M1:
    Gearbox = UsedWithDynamicTorqueLimitation
  M1/Gearbox/GearRatio:
    Input = 77
    Output = 2
  M1/Gearbox:
    MOTORGEAR_SPEED_MAX = 7500
    MOTORGEAR_TORQ_NOM = 424
    MOTORGEAR_TORQ_MAX = 424
    MOTORGEAR_INERTIA = 0.6
    MOTORGEAR_VISC_FRIC = 0.01
    MOTORGEAR_STAT_FRIC = 0.11
8LSA46.DB060S200-3-Q1_D4r1100R_5 : MotorSynchronous_any v2.2.1.0  [MT -> 8EI8X8HWT10.xxxx-1-Q1-Q2-Q3_D4r1100R_5.MT1]
  M1/MotorParameters:
    MOTOR_POLEPAIRS = 5
    MOTOR_SPEED_RATED = 6000
    MOTOR_SPEED_MAX = 12000
    MOTOR_VOLTAGE_RATED = 400
    MOTOR_CURR_RATED = 6.1
    MOTOR_CURR_STALL = 12.3
    MOTOR_CURR_MAX = 72.9
    MOTOR_TORQ_RATED = 5
    MOTOR_TORQ_STALL = 10
    MOTOR_TORQ_MAX = 38
    MOTOR_VOLTAGE_CONST = 49.22
    MOTOR_TORQ_CONST = 0.81
    MOTOR_STATOR_RESISTANCE = 0.48
    MOTOR_STATOR_INDUCTANCE = 4.35938
    MOTOR_INERTIA = 4.387
    VoltageLimitation = Used
  M1/MotorParameters/VoltageLimitation:
    MOTOR_UDC_MAX = 1000
  M1/MotorParameters/EncoderMounting:
    Angle = StoredOnEncoder
  M1/MotorParameters/TemperatureSensor:
    MOTOR_TEMPSENS_LIM = 130
    TemperatureSensorInterface = EncoderConnectorDigital
    MOTOR_TEMPSENS_PAR1 = 30
    MOTOR_TEMPSENS_PAR2 = 254
    MOTOR_TEMPSENS_PAR3 = -29.72
    MOTOR_TEMPSENS_PAR4 = -4.58
    MOTOR_TEMPSENS_PAR5 = 20.33
    MOTOR_TEMPSENS_PAR6 = 45.18
    MOTOR_TEMPSENS_PAR7 = 69.96
    MOTOR_TEMPSENS_PAR8 = 94.71
    MOTOR_TEMPSENS_PAR9 = 119.6
    MOTOR_TEMPSENS_PAR10 = 149.11
  M1/MotorParameters/TemperatureModel:
    MOTOR_WIND_TEMP_MAX = 110
  M1/MotorParameters/TemperatureModel/Calculation:
    MOTOR_WIND_CROSS_SECT = 1.765
    MOTOR_TAU_THERM = 2400
  M1:
    Brake = Used
  M1/Brake:
    MOTOR_BRAKE_CURR_RATED = 0.83
    MOTOR_BRAKE_TORQ_RATED = 8
    MOTOR_BRAKE_ON_TIME = 0.038
    MOTOR_BRAKE_OFF_TIME = 0.055
    MOTOR_BRAKE_INERTIA = 0.69
  M1/Encoder:
    MOTOR_ENCOD_ATTR = 1
    MOTOR_ENCOD_INERTIA = 0.026
    TemperatureSensor = Used
  M1/Encoder/TemperatureSensor:
    MOTOR_ENCOD_TEMP_LIM = 129
  M1:
    Gearbox = UsedWithDynamicTorqueLimitation
  M1/Gearbox/GearRatio:
    Input = 77
    Output = 2
  M1/Gearbox:
    MOTORGEAR_SPEED_MAX = 7500
    MOTORGEAR_TORQ_NOM = 424
    MOTORGEAR_TORQ_MAX = 424
    MOTORGEAR_INERTIA = 0.6
    MOTORGEAR_VISC_FRIC = 0.01
    MOTORGEAR_STAT_FRIC = 0.11
8LSA46.DB060S200-3-Q1_D4r1100R_6 : MotorSynchronous_any v2.2.1.0  [MT -> 8EI8X8HWT10.xxxx-1-Q1-Q2-Q3_D4r1100R_6.MT1]
  M1/MotorParameters:
    MOTOR_POLEPAIRS = 5
    MOTOR_SPEED_RATED = 6000
    MOTOR_SPEED_MAX = 12000
    MOTOR_VOLTAGE_RATED = 400
    MOTOR_CURR_RATED = 6.1
    MOTOR_CURR_STALL = 12.3
    MOTOR_CURR_MAX = 72.9
    MOTOR_TORQ_RATED = 5
    MOTOR_TORQ_STALL = 10
    MOTOR_TORQ_MAX = 38
    MOTOR_VOLTAGE_CONST = 49.22
    MOTOR_TORQ_CONST = 0.81
    MOTOR_STATOR_RESISTANCE = 0.48
    MOTOR_STATOR_INDUCTANCE = 4.35938
    MOTOR_INERTIA = 4.387
    VoltageLimitation = Used
  M1/MotorParameters/VoltageLimitation:
    MOTOR_UDC_MAX = 1000
  M1/MotorParameters/EncoderMounting:
    Angle = StoredOnEncoder
  M1/MotorParameters/TemperatureSensor:
    MOTOR_TEMPSENS_LIM = 130
    TemperatureSensorInterface = EncoderConnectorDigital
    MOTOR_TEMPSENS_PAR1 = 30
    MOTOR_TEMPSENS_PAR2 = 254
    MOTOR_TEMPSENS_PAR3 = -29.72
    MOTOR_TEMPSENS_PAR4 = -4.58
    MOTOR_TEMPSENS_PAR5 = 20.33
    MOTOR_TEMPSENS_PAR6 = 45.18
    MOTOR_TEMPSENS_PAR7 = 69.96
    MOTOR_TEMPSENS_PAR8 = 94.71
    MOTOR_TEMPSENS_PAR9 = 119.6
    MOTOR_TEMPSENS_PAR10 = 149.11
  M1/MotorParameters/TemperatureModel:
    MOTOR_WIND_TEMP_MAX = 110
  M1/MotorParameters/TemperatureModel/Calculation:
    MOTOR_WIND_CROSS_SECT = 1.765
    MOTOR_TAU_THERM = 2400
  M1:
    Brake = Used
  M1/Brake:
    MOTOR_BRAKE_CURR_RATED = 0.83
    MOTOR_BRAKE_TORQ_RATED = 8
    MOTOR_BRAKE_ON_TIME = 0.038
    MOTOR_BRAKE_OFF_TIME = 0.055
    MOTOR_BRAKE_INERTIA = 0.69
  M1/Encoder:
    MOTOR_ENCOD_ATTR = 1
    MOTOR_ENCOD_INERTIA = 0.026
    TemperatureSensor = Used
  M1/Encoder/TemperatureSensor:
    MOTOR_ENCOD_TEMP_LIM = 129
  M1:
    Gearbox = UsedWithDynamicTorqueLimitation
  M1/Gearbox/GearRatio:
    Input = 77
    Output = 2
  M1/Gearbox:
    MOTORGEAR_SPEED_MAX = 7500
    MOTORGEAR_TORQ_NOM = 424
    MOTORGEAR_TORQ_MAX = 424
    MOTORGEAR_INERTIA = 0.6
    MOTORGEAR_VISC_FRIC = 0.01
    MOTORGEAR_STAT_FRIC = 0.11
8LSA46.DB060S200-3-Q2_D4r1100R_1 : MotorSynchronous_any v2.2.1.0  [MT -> 8EI8X8HWT10.xxxx-1-Q1-Q2-Q3_D4r1100R_1.MT2]
  M1/MotorParameters:
    MOTOR_POLEPAIRS = 5
    MOTOR_SPEED_RATED = 6000
    MOTOR_SPEED_MAX = 12000
    MOTOR_VOLTAGE_RATED = 400
    MOTOR_CURR_RATED = 6.1
    MOTOR_CURR_STALL = 12.3
    MOTOR_CURR_MAX = 72.9
    MOTOR_TORQ_RATED = 5
    MOTOR_TORQ_STALL = 10
    MOTOR_TORQ_MAX = 38
    MOTOR_VOLTAGE_CONST = 49.22
    MOTOR_TORQ_CONST = 0.81
    MOTOR_STATOR_RESISTANCE = 0.48
    MOTOR_STATOR_INDUCTANCE = 4.35938
    MOTOR_INERTIA = 4.387
    VoltageLimitation = Used
  M1/MotorParameters/VoltageLimitation:
    MOTOR_UDC_MAX = 1000
  M1/MotorParameters/EncoderMounting:
    Angle = StoredOnEncoder
  M1/MotorParameters/TemperatureSensor:
    MOTOR_TEMPSENS_LIM = 130
    TemperatureSensorInterface = EncoderConnectorDigital
    MOTOR_TEMPSENS_PAR1 = 30
    MOTOR_TEMPSENS_PAR2 = 254
    MOTOR_TEMPSENS_PAR3 = -29.72
    MOTOR_TEMPSENS_PAR4 = -4.58
    MOTOR_TEMPSENS_PAR5 = 20.33
    MOTOR_TEMPSENS_PAR6 = 45.18
    MOTOR_TEMPSENS_PAR7 = 69.96
    MOTOR_TEMPSENS_PAR8 = 94.71
    MOTOR_TEMPSENS_PAR9 = 119.6
    MOTOR_TEMPSENS_PAR10 = 149.11
  M1/MotorParameters/TemperatureModel:
    MOTOR_WIND_TEMP_MAX = 110
  M1/MotorParameters/TemperatureModel/Calculation:
    MOTOR_WIND_CROSS_SECT = 1.765
    MOTOR_TAU_THERM = 2400
  M1:
    Brake = Used
  M1/Brake:
    MOTOR_BRAKE_CURR_RATED = 0.83
    MOTOR_BRAKE_TORQ_RATED = 8
    MOTOR_BRAKE_ON_TIME = 0.038
    MOTOR_BRAKE_OFF_TIME = 0.055
    MOTOR_BRAKE_INERTIA = 0.69
  M1/Encoder:
    MOTOR_ENCOD_ATTR = 1
    MOTOR_ENCOD_INERTIA = 0.026
    TemperatureSensor = Used
  M1/Encoder/TemperatureSensor:
    MOTOR_ENCOD_TEMP_LIM = 129
  M1:
    Gearbox = UsedWithDynamicTorqueLimitation
  M1/Gearbox/GearRatio:
    Input = 77
    Output = 2
  M1/Gearbox:
    MOTORGEAR_SPEED_MAX = 7500
    MOTORGEAR_TORQ_NOM = 424
    MOTORGEAR_TORQ_MAX = 424
    MOTORGEAR_INERTIA = 0.6
    MOTORGEAR_VISC_FRIC = 0.01
    MOTORGEAR_STAT_FRIC = 0.11
8LSA46.DB060S200-3-Q2_D4r1100R_2 : MotorSynchronous_any v2.2.1.0  [MT -> 8EI8X8HWT10.xxxx-1-Q1-Q2-Q3_D4r1100R_2.MT2]
  M1/MotorParameters:
    MOTOR_POLEPAIRS = 5
    MOTOR_SPEED_RATED = 6000
    MOTOR_SPEED_MAX = 12000
    MOTOR_VOLTAGE_RATED = 400
    MOTOR_CURR_RATED = 6.1
    MOTOR_CURR_STALL = 12.3
    MOTOR_CURR_MAX = 72.9
    MOTOR_TORQ_RATED = 5
    MOTOR_TORQ_STALL = 10
    MOTOR_TORQ_MAX = 38
    MOTOR_VOLTAGE_CONST = 49.22
    MOTOR_TORQ_CONST = 0.81
    MOTOR_STATOR_RESISTANCE = 0.48
    MOTOR_STATOR_INDUCTANCE = 4.35938
    MOTOR_INERTIA = 4.387
    VoltageLimitation = Used
  M1/MotorParameters/VoltageLimitation:
    MOTOR_UDC_MAX = 1000
  M1/MotorParameters/EncoderMounting:
    Angle = StoredOnEncoder
  M1/MotorParameters/TemperatureSensor:
    MOTOR_TEMPSENS_LIM = 130
    TemperatureSensorInterface = EncoderConnectorDigital
    MOTOR_TEMPSENS_PAR1 = 30
    MOTOR_TEMPSENS_PAR2 = 254
    MOTOR_TEMPSENS_PAR3 = -29.72
    MOTOR_TEMPSENS_PAR4 = -4.58
    MOTOR_TEMPSENS_PAR5 = 20.33
    MOTOR_TEMPSENS_PAR6 = 45.18
    MOTOR_TEMPSENS_PAR7 = 69.96
    MOTOR_TEMPSENS_PAR8 = 94.71
    MOTOR_TEMPSENS_PAR9 = 119.6
    MOTOR_TEMPSENS_PAR10 = 149.11
  M1/MotorParameters/TemperatureModel:
    MOTOR_WIND_TEMP_MAX = 110
  M1/MotorParameters/TemperatureModel/Calculation:
    MOTOR_WIND_CROSS_SECT = 1.765
    MOTOR_TAU_THERM = 2400
  M1:
    Brake = Used
  M1/Brake:
    MOTOR_BRAKE_CURR_RATED = 0.83
    MOTOR_BRAKE_TORQ_RATED = 8
    MOTOR_BRAKE_ON_TIME = 0.038
    MOTOR_BRAKE_OFF_TIME = 0.055
    MOTOR_BRAKE_INERTIA = 0.69
  M1/Encoder:
    MOTOR_ENCOD_ATTR = 1
    MOTOR_ENCOD_INERTIA = 0.026
    TemperatureSensor = Used
  M1/Encoder/TemperatureSensor:
    MOTOR_ENCOD_TEMP_LIM = 129
  M1:
    Gearbox = UsedWithDynamicTorqueLimitation
  M1/Gearbox/GearRatio:
    Input = 77
    Output = 2
  M1/Gearbox:
    MOTORGEAR_SPEED_MAX = 7500
    MOTORGEAR_TORQ_NOM = 424
    MOTORGEAR_TORQ_MAX = 424
    MOTORGEAR_INERTIA = 0.6
    MOTORGEAR_VISC_FRIC = 0.01
    MOTORGEAR_STAT_FRIC = 0.11
8LSA46.DB060S200-3-Q2_D4r1100R_3 : MotorSynchronous_any v2.2.1.0  [MT -> 8EI8X8HWT10.xxxx-1-Q1-Q2-Q3_D4r1100R_3.MT2]
  M1/MotorParameters:
    MOTOR_POLEPAIRS = 5
    MOTOR_SPEED_RATED = 6000
    MOTOR_SPEED_MAX = 12000
    MOTOR_VOLTAGE_RATED = 400
    MOTOR_CURR_RATED = 6.1
    MOTOR_CURR_STALL = 12.3
    MOTOR_CURR_MAX = 72.9
    MOTOR_TORQ_RATED = 5
    MOTOR_TORQ_STALL = 10
    MOTOR_TORQ_MAX = 38
    MOTOR_VOLTAGE_CONST = 49.22
    MOTOR_TORQ_CONST = 0.81
    MOTOR_STATOR_RESISTANCE = 0.48
    MOTOR_STATOR_INDUCTANCE = 4.35938
    MOTOR_INERTIA = 4.387
    VoltageLimitation = Used
  M1/MotorParameters/VoltageLimitation:
    MOTOR_UDC_MAX = 1000
  M1/MotorParameters/EncoderMounting:
    Angle = StoredOnEncoder
  M1/MotorParameters/TemperatureSensor:
    MOTOR_TEMPSENS_LIM = 130
    TemperatureSensorInterface = EncoderConnectorDigital
    MOTOR_TEMPSENS_PAR1 = 30
    MOTOR_TEMPSENS_PAR2 = 254
    MOTOR_TEMPSENS_PAR3 = -29.72
    MOTOR_TEMPSENS_PAR4 = -4.58
    MOTOR_TEMPSENS_PAR5 = 20.33
    MOTOR_TEMPSENS_PAR6 = 45.18
    MOTOR_TEMPSENS_PAR7 = 69.96
    MOTOR_TEMPSENS_PAR8 = 94.71
    MOTOR_TEMPSENS_PAR9 = 119.6
    MOTOR_TEMPSENS_PAR10 = 149.11
  M1/MotorParameters/TemperatureModel:
    MOTOR_WIND_TEMP_MAX = 110
  M1/MotorParameters/TemperatureModel/Calculation:
    MOTOR_WIND_CROSS_SECT = 1.765
    MOTOR_TAU_THERM = 2400
  M1:
    Brake = Used
  M1/Brake:
    MOTOR_BRAKE_CURR_RATED = 0.83
    MOTOR_BRAKE_TORQ_RATED = 8
    MOTOR_BRAKE_ON_TIME = 0.038
    MOTOR_BRAKE_OFF_TIME = 0.055
    MOTOR_BRAKE_INERTIA = 0.69
  M1/Encoder:
    MOTOR_ENCOD_ATTR = 1
    MOTOR_ENCOD_INERTIA = 0.026
    TemperatureSensor = Used
  M1/Encoder/TemperatureSensor:
    MOTOR_ENCOD_TEMP_LIM = 129
  M1:
    Gearbox = UsedWithDynamicTorqueLimitation
  M1/Gearbox/GearRatio:
    Input = 77
    Output = 2
  M1/Gearbox:
    MOTORGEAR_SPEED_MAX = 7500
    MOTORGEAR_TORQ_NOM = 424
    MOTORGEAR_TORQ_MAX = 424
    MOTORGEAR_INERTIA = 0.6
    MOTORGEAR_VISC_FRIC = 0.01
    MOTORGEAR_STAT_FRIC = 0.11
8LSA46.DB060S200-3-Q2_D4r1100R_4 : MotorSynchronous_any v2.2.1.0  [MT -> 8EI8X8HWT10.xxxx-1-Q1-Q2-Q3_D4r1100R_4.MT2]
  M1/MotorParameters:
    MOTOR_POLEPAIRS = 5
    MOTOR_SPEED_RATED = 6000
    MOTOR_SPEED_MAX = 12000
    MOTOR_VOLTAGE_RATED = 400
    MOTOR_CURR_RATED = 6.1
    MOTOR_CURR_STALL = 12.3
    MOTOR_CURR_MAX = 72.9
    MOTOR_TORQ_RATED = 5
    MOTOR_TORQ_STALL = 10
    MOTOR_TORQ_MAX = 38
    MOTOR_VOLTAGE_CONST = 49.22
    MOTOR_TORQ_CONST = 0.81
    MOTOR_STATOR_RESISTANCE = 0.48
    MOTOR_STATOR_INDUCTANCE = 4.35938
    MOTOR_INERTIA = 4.387
    VoltageLimitation = Used
  M1/MotorParameters/VoltageLimitation:
    MOTOR_UDC_MAX = 1000
  M1/MotorParameters/EncoderMounting:
    Angle = StoredOnEncoder
  M1/MotorParameters/TemperatureSensor:
    MOTOR_TEMPSENS_LIM = 130
    TemperatureSensorInterface = EncoderConnectorDigital
    MOTOR_TEMPSENS_PAR1 = 30
    MOTOR_TEMPSENS_PAR2 = 254
    MOTOR_TEMPSENS_PAR3 = -29.72
    MOTOR_TEMPSENS_PAR4 = -4.58
    MOTOR_TEMPSENS_PAR5 = 20.33
    MOTOR_TEMPSENS_PAR6 = 45.18
    MOTOR_TEMPSENS_PAR7 = 69.96
    MOTOR_TEMPSENS_PAR8 = 94.71
    MOTOR_TEMPSENS_PAR9 = 119.6
    MOTOR_TEMPSENS_PAR10 = 149.11
  M1/MotorParameters/TemperatureModel:
    MOTOR_WIND_TEMP_MAX = 110
  M1/MotorParameters/TemperatureModel/Calculation:
    MOTOR_WIND_CROSS_SECT = 1.765
    MOTOR_TAU_THERM = 2400
  M1:
    Brake = Used
  M1/Brake:
    MOTOR_BRAKE_CURR_RATED = 0.83
    MOTOR_BRAKE_TORQ_RATED = 8
    MOTOR_BRAKE_ON_TIME = 0.038
    MOTOR_BRAKE_OFF_TIME = 0.055
    MOTOR_BRAKE_INERTIA = 0.69
  M1/Encoder:
    MOTOR_ENCOD_ATTR = 1
    MOTOR_ENCOD_INERTIA = 0.026
    TemperatureSensor = Used
  M1/Encoder/TemperatureSensor:
    MOTOR_ENCOD_TEMP_LIM = 129
  M1:
    Gearbox = UsedWithDynamicTorqueLimitation
  M1/Gearbox/GearRatio:
    Input = 77
    Output = 2
  M1/Gearbox:
    MOTORGEAR_SPEED_MAX = 7500
    MOTORGEAR_TORQ_NOM = 424
    MOTORGEAR_TORQ_MAX = 424
    MOTORGEAR_INERTIA = 0.6
    MOTORGEAR_VISC_FRIC = 0.01
    MOTORGEAR_STAT_FRIC = 0.11
8LSA46.DB060S200-3-Q2_D4r1100R_5 : MotorSynchronous_any v2.2.1.0  [MT -> 8EI8X8HWT10.xxxx-1-Q1-Q2-Q3_D4r1100R_5.MT2]
  M1/MotorParameters:
    MOTOR_POLEPAIRS = 5
    MOTOR_SPEED_RATED = 6000
    MOTOR_SPEED_MAX = 12000
    MOTOR_VOLTAGE_RATED = 400
    MOTOR_CURR_RATED = 6.1
    MOTOR_CURR_STALL = 12.3
    MOTOR_CURR_MAX = 72.9
    MOTOR_TORQ_RATED = 5
    MOTOR_TORQ_STALL = 10
    MOTOR_TORQ_MAX = 38
    MOTOR_VOLTAGE_CONST = 49.22
    MOTOR_TORQ_CONST = 0.81
    MOTOR_STATOR_RESISTANCE = 0.48
    MOTOR_STATOR_INDUCTANCE = 4.35938
    MOTOR_INERTIA = 4.387
    VoltageLimitation = Used
  M1/MotorParameters/VoltageLimitation:
    MOTOR_UDC_MAX = 1000
  M1/MotorParameters/EncoderMounting:
    Angle = StoredOnEncoder
  M1/MotorParameters/TemperatureSensor:
    MOTOR_TEMPSENS_LIM = 130
    TemperatureSensorInterface = EncoderConnectorDigital
    MOTOR_TEMPSENS_PAR1 = 30
    MOTOR_TEMPSENS_PAR2 = 254
    MOTOR_TEMPSENS_PAR3 = -29.72
    MOTOR_TEMPSENS_PAR4 = -4.58
    MOTOR_TEMPSENS_PAR5 = 20.33
    MOTOR_TEMPSENS_PAR6 = 45.18
    MOTOR_TEMPSENS_PAR7 = 69.96
    MOTOR_TEMPSENS_PAR8 = 94.71
    MOTOR_TEMPSENS_PAR9 = 119.6
    MOTOR_TEMPSENS_PAR10 = 149.11
  M1/MotorParameters/TemperatureModel:
    MOTOR_WIND_TEMP_MAX = 110
  M1/MotorParameters/TemperatureModel/Calculation:
    MOTOR_WIND_CROSS_SECT = 1.765
    MOTOR_TAU_THERM = 2400
  M1:
    Brake = Used
  M1/Brake:
    MOTOR_BRAKE_CURR_RATED = 0.83
    MOTOR_BRAKE_TORQ_RATED = 8
    MOTOR_BRAKE_ON_TIME = 0.038
    MOTOR_BRAKE_OFF_TIME = 0.055
    MOTOR_BRAKE_INERTIA = 0.69
  M1/Encoder:
    MOTOR_ENCOD_ATTR = 1
    MOTOR_ENCOD_INERTIA = 0.026
    TemperatureSensor = Used
  M1/Encoder/TemperatureSensor:
    MOTOR_ENCOD_TEMP_LIM = 129
  M1:
    Gearbox = UsedWithDynamicTorqueLimitation
  M1/Gearbox/GearRatio:
    Input = 77
    Output = 2
  M1/Gearbox:
    MOTORGEAR_SPEED_MAX = 7500
    MOTORGEAR_TORQ_NOM = 424
    MOTORGEAR_TORQ_MAX = 424
    MOTORGEAR_INERTIA = 0.6
    MOTORGEAR_VISC_FRIC = 0.01
    MOTORGEAR_STAT_FRIC = 0.11
8LSA46.DB060S200-3-Q2_D4r1100R_6 : MotorSynchronous_any v2.2.1.0  [MT -> 8EI8X8HWT10.xxxx-1-Q1-Q2-Q3_D4r1100R_6.MT2]
  M1/MotorParameters:
    MOTOR_POLEPAIRS = 5
    MOTOR_SPEED_RATED = 6000
    MOTOR_SPEED_MAX = 12000
    MOTOR_VOLTAGE_RATED = 400
    MOTOR_CURR_RATED = 6.1
    MOTOR_CURR_STALL = 12.3
    MOTOR_CURR_MAX = 72.9
    MOTOR_TORQ_RATED = 5
    MOTOR_TORQ_STALL = 10
    MOTOR_TORQ_MAX = 38
    MOTOR_VOLTAGE_CONST = 49.22
    MOTOR_TORQ_CONST = 0.81
    MOTOR_STATOR_RESISTANCE = 0.48
    MOTOR_STATOR_INDUCTANCE = 4.35938
    MOTOR_INERTIA = 4.387
    VoltageLimitation = Used
  M1/MotorParameters/VoltageLimitation:
    MOTOR_UDC_MAX = 1000
  M1/MotorParameters/EncoderMounting:
    Angle = StoredOnEncoder
  M1/MotorParameters/TemperatureSensor:
    MOTOR_TEMPSENS_LIM = 130
    TemperatureSensorInterface = EncoderConnectorDigital
    MOTOR_TEMPSENS_PAR1 = 30
    MOTOR_TEMPSENS_PAR2 = 254
    MOTOR_TEMPSENS_PAR3 = -29.72
    MOTOR_TEMPSENS_PAR4 = -4.58
    MOTOR_TEMPSENS_PAR5 = 20.33
    MOTOR_TEMPSENS_PAR6 = 45.18
    MOTOR_TEMPSENS_PAR7 = 69.96
    MOTOR_TEMPSENS_PAR8 = 94.71
    MOTOR_TEMPSENS_PAR9 = 119.6
    MOTOR_TEMPSENS_PAR10 = 149.11
  M1/MotorParameters/TemperatureModel:
    MOTOR_WIND_TEMP_MAX = 110
  M1/MotorParameters/TemperatureModel/Calculation:
    MOTOR_WIND_CROSS_SECT = 1.765
    MOTOR_TAU_THERM = 2400
  M1:
    Brake = Used
  M1/Brake:
    MOTOR_BRAKE_CURR_RATED = 0.83
    MOTOR_BRAKE_TORQ_RATED = 8
    MOTOR_BRAKE_ON_TIME = 0.038
    MOTOR_BRAKE_OFF_TIME = 0.055
    MOTOR_BRAKE_INERTIA = 0.69
  M1/Encoder:
    MOTOR_ENCOD_ATTR = 1
    MOTOR_ENCOD_INERTIA = 0.026
    TemperatureSensor = Used
  M1/Encoder/TemperatureSensor:
    MOTOR_ENCOD_TEMP_LIM = 129
  M1:
    Gearbox = UsedWithDynamicTorqueLimitation
  M1/Gearbox/GearRatio:
    Input = 77
    Output = 2
  M1/Gearbox:
    MOTORGEAR_SPEED_MAX = 7500
    MOTORGEAR_TORQ_NOM = 424
    MOTORGEAR_TORQ_MAX = 424
    MOTORGEAR_INERTIA = 0.6
    MOTORGEAR_VISC_FRIC = 0.01
    MOTORGEAR_STAT_FRIC = 0.11
8LSA46.DB060S200-3-Q3_D4r1100R_1 : MotorSynchronous_any v2.2.1.0  [MT -> 8EI8X8HWT10.xxxx-1-Q1-Q2-Q3_D4r1100R_1.MT3]
  M1/MotorParameters:
    MOTOR_POLEPAIRS = 5
    MOTOR_SPEED_RATED = 6000
    MOTOR_SPEED_MAX = 12000
    MOTOR_VOLTAGE_RATED = 400
    MOTOR_CURR_RATED = 6.1
    MOTOR_CURR_STALL = 12.3
    MOTOR_CURR_MAX = 72.9
    MOTOR_TORQ_RATED = 5
    MOTOR_TORQ_STALL = 10
    MOTOR_TORQ_MAX = 38
    MOTOR_VOLTAGE_CONST = 49.22
    MOTOR_TORQ_CONST = 0.81
    MOTOR_STATOR_RESISTANCE = 0.48
    MOTOR_STATOR_INDUCTANCE = 4.35938
    MOTOR_INERTIA = 4.387
    VoltageLimitation = Used
  M1/MotorParameters/VoltageLimitation:
    MOTOR_UDC_MAX = 1000
  M1/MotorParameters/EncoderMounting:
    Angle = StoredOnEncoder
  M1/MotorParameters/TemperatureSensor:
    MOTOR_TEMPSENS_LIM = 130
    TemperatureSensorInterface = EncoderConnectorDigital
    MOTOR_TEMPSENS_PAR1 = 30
    MOTOR_TEMPSENS_PAR2 = 254
    MOTOR_TEMPSENS_PAR3 = -29.72
    MOTOR_TEMPSENS_PAR4 = -4.58
    MOTOR_TEMPSENS_PAR5 = 20.33
    MOTOR_TEMPSENS_PAR6 = 45.18
    MOTOR_TEMPSENS_PAR7 = 69.96
    MOTOR_TEMPSENS_PAR8 = 94.71
    MOTOR_TEMPSENS_PAR9 = 119.6
    MOTOR_TEMPSENS_PAR10 = 149.11
  M1/MotorParameters/TemperatureModel:
    MOTOR_WIND_TEMP_MAX = 110
  M1/MotorParameters/TemperatureModel/Calculation:
    MOTOR_WIND_CROSS_SECT = 1.765
    MOTOR_TAU_THERM = 2400
  M1:
    Brake = Used
  M1/Brake:
    MOTOR_BRAKE_CURR_RATED = 0.83
    MOTOR_BRAKE_TORQ_RATED = 8
    MOTOR_BRAKE_ON_TIME = 0.038
    MOTOR_BRAKE_OFF_TIME = 0.055
    MOTOR_BRAKE_INERTIA = 0.69
  M1/Encoder:
    MOTOR_ENCOD_ATTR = 1
    MOTOR_ENCOD_INERTIA = 0.026
    TemperatureSensor = Used
  M1/Encoder/TemperatureSensor:
    MOTOR_ENCOD_TEMP_LIM = 129
  M1:
    Gearbox = UsedWithDynamicTorqueLimitation
  M1/Gearbox/GearRatio:
    Input = 77
    Output = 2
  M1/Gearbox:
    MOTORGEAR_SPEED_MAX = 7500
    MOTORGEAR_TORQ_NOM = 424
    MOTORGEAR_TORQ_MAX = 424
    MOTORGEAR_INERTIA = 0.6
    MOTORGEAR_VISC_FRIC = 0.01
    MOTORGEAR_STAT_FRIC = 0.11
8LSA46.DB060S200-3-Q3_D4r1100R_2 : MotorSynchronous_any v2.2.1.0  [MT -> 8EI8X8HWT10.xxxx-1-Q1-Q2-Q3_D4r1100R_2.MT3]
  M1/MotorParameters:
    MOTOR_POLEPAIRS = 5
    MOTOR_SPEED_RATED = 6000
    MOTOR_SPEED_MAX = 12000
    MOTOR_VOLTAGE_RATED = 400
    MOTOR_CURR_RATED = 6.1
    MOTOR_CURR_STALL = 12.3
    MOTOR_CURR_MAX = 72.9
    MOTOR_TORQ_RATED = 5
    MOTOR_TORQ_STALL = 10
    MOTOR_TORQ_MAX = 38
    MOTOR_VOLTAGE_CONST = 49.22
    MOTOR_TORQ_CONST = 0.81
    MOTOR_STATOR_RESISTANCE = 0.48
    MOTOR_STATOR_INDUCTANCE = 4.35938
    MOTOR_INERTIA = 4.387
    VoltageLimitation = Used
  M1/MotorParameters/VoltageLimitation:
    MOTOR_UDC_MAX = 1000
  M1/MotorParameters/EncoderMounting:
    Angle = StoredOnEncoder
  M1/MotorParameters/TemperatureSensor:
    MOTOR_TEMPSENS_LIM = 130
    TemperatureSensorInterface = EncoderConnectorDigital
    MOTOR_TEMPSENS_PAR1 = 30
    MOTOR_TEMPSENS_PAR2 = 254
    MOTOR_TEMPSENS_PAR3 = -29.72
    MOTOR_TEMPSENS_PAR4 = -4.58
    MOTOR_TEMPSENS_PAR5 = 20.33
    MOTOR_TEMPSENS_PAR6 = 45.18
    MOTOR_TEMPSENS_PAR7 = 69.96
    MOTOR_TEMPSENS_PAR8 = 94.71
    MOTOR_TEMPSENS_PAR9 = 119.6
    MOTOR_TEMPSENS_PAR10 = 149.11
  M1/MotorParameters/TemperatureModel:
    MOTOR_WIND_TEMP_MAX = 110
  M1/MotorParameters/TemperatureModel/Calculation:
    MOTOR_WIND_CROSS_SECT = 1.765
    MOTOR_TAU_THERM = 2400
  M1:
    Brake = Used
  M1/Brake:
    MOTOR_BRAKE_CURR_RATED = 0.83
    MOTOR_BRAKE_TORQ_RATED = 8
    MOTOR_BRAKE_ON_TIME = 0.038
    MOTOR_BRAKE_OFF_TIME = 0.055
    MOTOR_BRAKE_INERTIA = 0.69
  M1/Encoder:
    MOTOR_ENCOD_ATTR = 1
    MOTOR_ENCOD_INERTIA = 0.026
    TemperatureSensor = Used
  M1/Encoder/TemperatureSensor:
    MOTOR_ENCOD_TEMP_LIM = 129
  M1:
    Gearbox = UsedWithDynamicTorqueLimitation
  M1/Gearbox/GearRatio:
    Input = 77
    Output = 2
  M1/Gearbox:
    MOTORGEAR_SPEED_MAX = 7500
    MOTORGEAR_TORQ_NOM = 424
    MOTORGEAR_TORQ_MAX = 424
    MOTORGEAR_INERTIA = 0.6
    MOTORGEAR_VISC_FRIC = 0.01
    MOTORGEAR_STAT_FRIC = 0.11
8LSA46.DB060S200-3-Q3_D4r1100R_3 : MotorSynchronous_any v2.2.1.0  [MT -> 8EI8X8HWT10.xxxx-1-Q1-Q2-Q3_D4r1100R_3.MT3]
  M1/MotorParameters:
    MOTOR_POLEPAIRS = 5
    MOTOR_SPEED_RATED = 6000
    MOTOR_SPEED_MAX = 12000
    MOTOR_VOLTAGE_RATED = 400
    MOTOR_CURR_RATED = 6.1
    MOTOR_CURR_STALL = 12.3
    MOTOR_CURR_MAX = 72.9
    MOTOR_TORQ_RATED = 5
    MOTOR_TORQ_STALL = 10
    MOTOR_TORQ_MAX = 38
    MOTOR_VOLTAGE_CONST = 49.22
    MOTOR_TORQ_CONST = 0.81
    MOTOR_STATOR_RESISTANCE = 0.48
    MOTOR_STATOR_INDUCTANCE = 4.35938
    MOTOR_INERTIA = 4.387
    VoltageLimitation = Used
  M1/MotorParameters/VoltageLimitation:
    MOTOR_UDC_MAX = 1000
  M1/MotorParameters/EncoderMounting:
    Angle = StoredOnEncoder
  M1/MotorParameters/TemperatureSensor:
    MOTOR_TEMPSENS_LIM = 130
    TemperatureSensorInterface = EncoderConnectorDigital
    MOTOR_TEMPSENS_PAR1 = 30
    MOTOR_TEMPSENS_PAR2 = 254
    MOTOR_TEMPSENS_PAR3 = -29.72
    MOTOR_TEMPSENS_PAR4 = -4.58
    MOTOR_TEMPSENS_PAR5 = 20.33
    MOTOR_TEMPSENS_PAR6 = 45.18
    MOTOR_TEMPSENS_PAR7 = 69.96
    MOTOR_TEMPSENS_PAR8 = 94.71
    MOTOR_TEMPSENS_PAR9 = 119.6
    MOTOR_TEMPSENS_PAR10 = 149.11
  M1/MotorParameters/TemperatureModel:
    MOTOR_WIND_TEMP_MAX = 110
  M1/MotorParameters/TemperatureModel/Calculation:
    MOTOR_WIND_CROSS_SECT = 1.765
    MOTOR_TAU_THERM = 2400
  M1:
    Brake = Used
  M1/Brake:
    MOTOR_BRAKE_CURR_RATED = 0.83
    MOTOR_BRAKE_TORQ_RATED = 8
    MOTOR_BRAKE_ON_TIME = 0.038
    MOTOR_BRAKE_OFF_TIME = 0.055
    MOTOR_BRAKE_INERTIA = 0.69
  M1/Encoder:
    MOTOR_ENCOD_ATTR = 1
    MOTOR_ENCOD_INERTIA = 0.026
    TemperatureSensor = Used
  M1/Encoder/TemperatureSensor:
    MOTOR_ENCOD_TEMP_LIM = 129
  M1:
    Gearbox = UsedWithDynamicTorqueLimitation
  M1/Gearbox/GearRatio:
    Input = 77
    Output = 2
  M1/Gearbox:
    MOTORGEAR_SPEED_MAX = 7500
    MOTORGEAR_TORQ_NOM = 424
    MOTORGEAR_TORQ_MAX = 424
    MOTORGEAR_INERTIA = 0.6
    MOTORGEAR_VISC_FRIC = 0.01
    MOTORGEAR_STAT_FRIC = 0.11
8LSA46.DB060S200-3-Q3_D4r1100R_4 : MotorSynchronous_any v2.2.1.0  [MT -> 8EI8X8HWT10.xxxx-1-Q1-Q2-Q3_D4r1100R_4.MT3]
  M1/MotorParameters:
    MOTOR_POLEPAIRS = 5
    MOTOR_SPEED_RATED = 6000
    MOTOR_SPEED_MAX = 12000
    MOTOR_VOLTAGE_RATED = 400
    MOTOR_CURR_RATED = 6.1
    MOTOR_CURR_STALL = 12.3
    MOTOR_CURR_MAX = 72.9
    MOTOR_TORQ_RATED = 5
    MOTOR_TORQ_STALL = 10
    MOTOR_TORQ_MAX = 38
    MOTOR_VOLTAGE_CONST = 49.22
    MOTOR_TORQ_CONST = 0.81
    MOTOR_STATOR_RESISTANCE = 0.48
    MOTOR_STATOR_INDUCTANCE = 4.35938
    MOTOR_INERTIA = 4.387
    VoltageLimitation = Used
  M1/MotorParameters/VoltageLimitation:
    MOTOR_UDC_MAX = 1000
  M1/MotorParameters/EncoderMounting:
    Angle = StoredOnEncoder
  M1/MotorParameters/TemperatureSensor:
    MOTOR_TEMPSENS_LIM = 130
    TemperatureSensorInterface = EncoderConnectorDigital
    MOTOR_TEMPSENS_PAR1 = 30
    MOTOR_TEMPSENS_PAR2 = 254
    MOTOR_TEMPSENS_PAR3 = -29.72
    MOTOR_TEMPSENS_PAR4 = -4.58
    MOTOR_TEMPSENS_PAR5 = 20.33
    MOTOR_TEMPSENS_PAR6 = 45.18
    MOTOR_TEMPSENS_PAR7 = 69.96
    MOTOR_TEMPSENS_PAR8 = 94.71
    MOTOR_TEMPSENS_PAR9 = 119.6
    MOTOR_TEMPSENS_PAR10 = 149.11
  M1/MotorParameters/TemperatureModel:
    MOTOR_WIND_TEMP_MAX = 110
  M1/MotorParameters/TemperatureModel/Calculation:
    MOTOR_WIND_CROSS_SECT = 1.765
    MOTOR_TAU_THERM = 2400
  M1:
    Brake = Used
  M1/Brake:
    MOTOR_BRAKE_CURR_RATED = 0.83
    MOTOR_BRAKE_TORQ_RATED = 8
    MOTOR_BRAKE_ON_TIME = 0.038
    MOTOR_BRAKE_OFF_TIME = 0.055
    MOTOR_BRAKE_INERTIA = 0.69
  M1/Encoder:
    MOTOR_ENCOD_ATTR = 1
    MOTOR_ENCOD_INERTIA = 0.026
    TemperatureSensor = Used
  M1/Encoder/TemperatureSensor:
    MOTOR_ENCOD_TEMP_LIM = 129
  M1:
    Gearbox = UsedWithDynamicTorqueLimitation
  M1/Gearbox/GearRatio:
    Input = 77
    Output = 2
  M1/Gearbox:
    MOTORGEAR_SPEED_MAX = 7500
    MOTORGEAR_TORQ_NOM = 424
    MOTORGEAR_TORQ_MAX = 424
    MOTORGEAR_INERTIA = 0.6
    MOTORGEAR_VISC_FRIC = 0.01
    MOTORGEAR_STAT_FRIC = 0.11
8LSA46.DB060S200-3-Q3_D4r1100R_5 : MotorSynchronous_any v2.2.1.0  [MT -> 8EI8X8HWT10.xxxx-1-Q1-Q2-Q3_D4r1100R_5.MT3]
  M1/MotorParameters:
    MOTOR_POLEPAIRS = 5
    MOTOR_SPEED_RATED = 6000
    MOTOR_SPEED_MAX = 12000
    MOTOR_VOLTAGE_RATED = 400
    MOTOR_CURR_RATED = 6.1
    MOTOR_CURR_STALL = 12.3
    MOTOR_CURR_MAX = 72.9
    MOTOR_TORQ_RATED = 5
    MOTOR_TORQ_STALL = 10
    MOTOR_TORQ_MAX = 38
    MOTOR_VOLTAGE_CONST = 49.22
    MOTOR_TORQ_CONST = 0.81
    MOTOR_STATOR_RESISTANCE = 0.48
    MOTOR_STATOR_INDUCTANCE = 4.35938
    MOTOR_INERTIA = 4.387
    VoltageLimitation = Used
  M1/MotorParameters/VoltageLimitation:
    MOTOR_UDC_MAX = 1000
  M1/MotorParameters/EncoderMounting:
    Angle = StoredOnEncoder
  M1/MotorParameters/TemperatureSensor:
    MOTOR_TEMPSENS_LIM = 130
    TemperatureSensorInterface = EncoderConnectorDigital
    MOTOR_TEMPSENS_PAR1 = 30
    MOTOR_TEMPSENS_PAR2 = 254
    MOTOR_TEMPSENS_PAR3 = -29.72
    MOTOR_TEMPSENS_PAR4 = -4.58
    MOTOR_TEMPSENS_PAR5 = 20.33
    MOTOR_TEMPSENS_PAR6 = 45.18
    MOTOR_TEMPSENS_PAR7 = 69.96
    MOTOR_TEMPSENS_PAR8 = 94.71
    MOTOR_TEMPSENS_PAR9 = 119.6
    MOTOR_TEMPSENS_PAR10 = 149.11
  M1/MotorParameters/TemperatureModel:
    MOTOR_WIND_TEMP_MAX = 110
  M1/MotorParameters/TemperatureModel/Calculation:
    MOTOR_WIND_CROSS_SECT = 1.765
    MOTOR_TAU_THERM = 2400
  M1:
    Brake = Used
  M1/Brake:
    MOTOR_BRAKE_CURR_RATED = 0.83
    MOTOR_BRAKE_TORQ_RATED = 8
    MOTOR_BRAKE_ON_TIME = 0.038
    MOTOR_BRAKE_OFF_TIME = 0.055
    MOTOR_BRAKE_INERTIA = 0.69
  M1/Encoder:
    MOTOR_ENCOD_ATTR = 1
    MOTOR_ENCOD_INERTIA = 0.026
    TemperatureSensor = Used
  M1/Encoder/TemperatureSensor:
    MOTOR_ENCOD_TEMP_LIM = 129
  M1:
    Gearbox = UsedWithDynamicTorqueLimitation
  M1/Gearbox/GearRatio:
    Input = 77
    Output = 2
  M1/Gearbox:
    MOTORGEAR_SPEED_MAX = 7500
    MOTORGEAR_TORQ_NOM = 424
    MOTORGEAR_TORQ_MAX = 424
    MOTORGEAR_INERTIA = 0.6
    MOTORGEAR_VISC_FRIC = 0.01
    MOTORGEAR_STAT_FRIC = 0.11
8LSA46.DB060S200-3-Q3_D4r1100R_6 : MotorSynchronous_any v2.2.1.0  [MT -> 8EI8X8HWT10.xxxx-1-Q1-Q2-Q3_D4r1100R_6.MT3]
  M1/MotorParameters:
    MOTOR_POLEPAIRS = 5
    MOTOR_SPEED_RATED = 6000
    MOTOR_SPEED_MAX = 12000
    MOTOR_VOLTAGE_RATED = 400
    MOTOR_CURR_RATED = 6.1
    MOTOR_CURR_STALL = 12.3
    MOTOR_CURR_MAX = 72.9
    MOTOR_TORQ_RATED = 5
    MOTOR_TORQ_STALL = 10
    MOTOR_TORQ_MAX = 38
    MOTOR_VOLTAGE_CONST = 49.22
    MOTOR_TORQ_CONST = 0.81
    MOTOR_STATOR_RESISTANCE = 0.48
    MOTOR_STATOR_INDUCTANCE = 4.35938
    MOTOR_INERTIA = 4.387
    VoltageLimitation = Used
  M1/MotorParameters/VoltageLimitation:
    MOTOR_UDC_MAX = 1000
  M1/MotorParameters/EncoderMounting:
    Angle = StoredOnEncoder
  M1/MotorParameters/TemperatureSensor:
    MOTOR_TEMPSENS_LIM = 130
    TemperatureSensorInterface = EncoderConnectorDigital
    MOTOR_TEMPSENS_PAR1 = 30
    MOTOR_TEMPSENS_PAR2 = 254
    MOTOR_TEMPSENS_PAR3 = -29.72
    MOTOR_TEMPSENS_PAR4 = -4.58
    MOTOR_TEMPSENS_PAR5 = 20.33
    MOTOR_TEMPSENS_PAR6 = 45.18
    MOTOR_TEMPSENS_PAR7 = 69.96
    MOTOR_TEMPSENS_PAR8 = 94.71
    MOTOR_TEMPSENS_PAR9 = 119.6
    MOTOR_TEMPSENS_PAR10 = 149.11
  M1/MotorParameters/TemperatureModel:
    MOTOR_WIND_TEMP_MAX = 110
  M1/MotorParameters/TemperatureModel/Calculation:
    MOTOR_WIND_CROSS_SECT = 1.765
    MOTOR_TAU_THERM = 2400
  M1:
    Brake = Used
  M1/Brake:
    MOTOR_BRAKE_CURR_RATED = 0.83
    MOTOR_BRAKE_TORQ_RATED = 8
    MOTOR_BRAKE_ON_TIME = 0.038
    MOTOR_BRAKE_OFF_TIME = 0.055
    MOTOR_BRAKE_INERTIA = 0.69
  M1/Encoder:
    MOTOR_ENCOD_ATTR = 1
    MOTOR_ENCOD_INERTIA = 0.026
    TemperatureSensor = Used
  M1/Encoder/TemperatureSensor:
    MOTOR_ENCOD_TEMP_LIM = 129
  M1:
    Gearbox = UsedWithDynamicTorqueLimitation
  M1/Gearbox/GearRatio:
    Input = 77
    Output = 2
  M1/Gearbox:
    MOTORGEAR_SPEED_MAX = 7500
    MOTORGEAR_TORQ_NOM = 424
    MOTORGEAR_TORQ_MAX = 424
    MOTORGEAR_INERTIA = 0.6
    MOTORGEAR_VISC_FRIC = 0.01
    MOTORGEAR_STAT_FRIC = 0.11
```
